C03632=1090.259,178.898,430.027,176.034,19.768,152.995
C03633=1090.254,178.648,430.050,176.031,19.767,152.995
C03634=1090.248,178.399,430.073,176.028,19.766,152.995
C03635=1090.242,178.150,430.094,176.025,19.765,152.995
C03636=1090.237,177.901,430.116,176.023,19.764,152.995
C03637=1090.232,177.652,430.139,176.020,19.763,152.996
C03638=1090.225,177.403,430.161,176.017,19.762,152.996
C03639=1090.220,177.155,430.183,176.014,19.761,152.996
C03640=1090.215,176.906,430.206,176.012,19.760,152.997
C03641=1090.209,176.656,430.227,176.009,19.759,152.997
C03642=1090.203,176.407,430.250,176.006,19.758,152.997
C03643=1090.197,176.131,430.274,176.003,19.756,152.997
C03644=1090.191,175.854,430.299,176.001,19.755,152.997
C03645=1090.184,175.577,430.323,175.997,19.753,152.998
C03646=1090.178,175.300,430.348,175.994,19.752,152.998
C03647=1090.172,175.051,430.370,175.992,19.751,152.998
C03648=1090.167,174.803,430.393,175.989,19.750,152.998
C03649=1090.162,174.553,430.415,175.986,19.749,152.999
C03650=1090.155,174.304,430.437,175.983,19.748,152.999
C03651=1090.151,174.055,430.458,175.981,19.747,152.999
C03652=1090.144,173.806,430.481,175.978,19.746,152.999
C03653=1090.139,173.557,430.503,175.975,19.745,153.000
C03654=1090.134,173.308,430.525,175.972,19.744,153.000
C03655=1090.128,173.059,430.546,175.970,19.742,153.000
C03656=1090.123,172.811,430.569,175.967,19.741,153.000
C03657=1090.116,172.561,430.591,175.965,19.740,153.000
C03658=1090.111,172.312,430.613,175.962,19.739,153.001
C03659=1090.106,172.063,430.634,175.960,19.738,153.001
C03660=1090.100,171.814,430.656,175.957,19.737,153.001
C03661=1090.095,171.565,430.678,175.954,19.736,153.001
C03662=1090.089,171.317,430.701,175.952,19.734,153.001
C03663=1090.084,171.068,430.722,175.949,19.733,153.002
C03664=1090.078,170.819,430.744,175.946,19.732,153.002
C03665=1090.073,170.570,430.766,175.943,19.731,153.002
C03666=1090.067,170.321,430.788,175.941,19.730,153.002
C03667=1090.061,170.071,430.810,175.938,19.729,153.003
C03668=1090.056,169.822,430.831,175.935,19.728,153.003
C03669=1090.050,169.573,430.853,175.933,19.726,153.003
C03670=1090.045,169.324,430.875,175.930,19.725,153.003
C03671=1090.039,169.076,430.898,175.927,19.724,153.004
C03672=1090.034,168.827,430.919,175.925,19.722,153.004
C03673=1090.028,168.578,430.941,175.923,19.722,153.004
C03674=1090.023,168.329,430.962,175.920,19.720,153.004
C03675=1090.017,168.080,430.985,175.917,19.719,153.004
C03676=1090.012,167.831,431.006,175.915,19.718,153.004
C03677=1090.006,167.582,431.028,175.912,19.717,153.005
C03678=1090.001,167.333,431.049,175.909,19.716,153.005
C03679=1089.995,167.083,431.072,175.906,19.715,153.005
C03680=1089.990,166.835,431.093,175.904,19.713,153.005
C03681=1089.984,166.586,431.114,175.901,19.712,153.005
C03682=1089.979,166.336,431.136,175.899,19.711,153.006
C03683=1089.973,166.088,431.157,175.896,19.710,153.006
C03684=1089.968,165.838,431.179,175.893,19.708,153.006
C03685=1089.962,165.590,431.200,175.891,19.707,153.006
C03686=1089.957,165.340,431.223,175.889,19.707,153.006
C03687=1089.951,165.092,431.244,175.886,19.705,153.007
C03688=1089.946,164.842,431.266,175.883,19.704,153.007
C03689=1089.940,164.594,431.287,175.881,19.702,153.007
C03690=1089.935,164.345,431.309,175.878,19.701,153.007
C03691=1089.930,164.095,431.330,175.875,19.700,153.007
C03692=1089.924,163.847,431.351,175.873,19.699,153.008
C03693=1089.919,163.597,431.374,175.870,19.697,153.008
C03694=1089.913,163.349,431.395,175.867,19.696,153.008
C03695=1089.908,163.100,431.416,175.865,19.695,153.008
C03696=1089.902,162.851,431.438,175.863,19.694,153.008
C03697=1089.897,162.601,431.459,175.860,19.693,153.008
C03698=1089.892,162.353,431.481,175.858,19.692,153.009
C03699=1089.886,162.103,431.502,175.855,19.690,153.009
C03700=1089.880,161.855,431.524,175.852,19.689,153.009
C03701=1089.876,161.606,431.545,175.850,19.688,153.009
C03702=1089.870,161.356,431.567,175.847,19.687,153.009
C03703=1089.864,161.108,431.588,175.844,19.685,153.010
C03704=1089.858,160.858,431.609,175.842,19.684,153.010
C03705=1089.853,160.609,431.630,175.840,19.683,153.010
C03706=1089.847,160.360,431.652,175.837,19.682,153.010
C03707=1089.841,160.083,431.676,175.834,19.680,153.010
C03708=1089.835,159.806,431.700,175.831,19.679,153.011
C03709=1089.829,159.528,431.723,175.828,19.678,153.011
C03710=1089.822,159.251,431.747,175.825,19.677,153.011
C03711=1089.817,159.002,431.768,175.823,19.675,153.011
C03712=1089.811,158.754,431.789,175.820,19.674,153.011
C03713=1089.806,158.504,431.810,175.818,19.673,153.012
C03714=1089.800,158.255,431.831,175.815,19.672,153.012
C03715=1089.794,158.005,431.852,175.813,19.671,153.012
C03716=1089.789,157.757,431.873,175.810,19.670,153.012
C03717=1089.783,157.508,431.895,175.808,19.668,153.012
C03718=1089.777,157.259,431.916,175.805,19.667,153.013
C03719=1089.772,157.010,431.937,175.802,19.666,153.013
C03720=1089.767,156.761,431.958,175.800,19.664,153.013
C03721=1089.761,156.511,431.980,175.797,19.663,153.013
C03722=1089.756,156.262,432.000,175.795,19.662,153.013
C03723=1089.750,156.014,432.021,175.793,19.661,153.013
C03724=1089.744,155.764,432.042,175.790,19.660,153.014
C03725=1089.739,155.516,432.064,175.787,19.658,153.014
C03726=1089.733,155.266,432.084,175.785,19.657,153.014
C03727=1089.727,155.017,432.106,175.782,19.656,153.014
C03728=1089.722,154.768,432.126,175.779,19.655,153.014
C03729=1089.716,154.520,432.148,175.778,19.654,153.015
C03730=1089.711,154.270,432.169,175.775,19.653,153.015
C03731=1089.705,154.021,432.190,175.772,19.651,153.015
C03732=1089.700,153.772,432.210,175.769,19.650,153.015
C03733=1089.694,153.524,432.232,175.767,19.649,153.015
C03734=1089.688,153.274,432.253,175.764,19.648,153.016
C03735=1089.682,153.025,432.273,175.762,19.647,153.016
C03736=1089.677,152.776,432.294,175.760,19.646,153.016
C03737=1089.671,152.527,432.315,175.757,19.644,153.016
C03738=1089.666,152.278,432.335,175.755,19.642,153.016
C03739=1089.660,152.029,432.357,175.752,19.641,153.016
C03740=1089.655,151.780,432.377,175.749,19.640,153.017
C03741=1089.649,151.530,432.398,175.747,19.639,153.017
C03742=1089.643,151.282,432.419,175.745,19.638,153.017
C03743=1089.638,151.032,432.440,175.742,19.636,153.017
C03744=1089.633,150.783,432.460,175.739,19.635,153.017
C03745=1089.627,150.534,432.482,175.737,19.634,153.017
C03746=1089.621,150.285,432.502,175.734,19.633,153.018
C03747=1089.615,150.036,432.523,175.732,19.632,153.018
C03748=1089.610,149.788,432.544,175.730,19.630,153.018
C03749=1089.605,149.539,432.564,175.727,19.629,153.018
C03750=1089.599,149.289,432.585,175.725,19.628,153.018
C03751=1089.594,149.040,432.606,175.722,19.626,153.018
C03752=1089.588,148.791,432.627,175.719,19.625,153.019
C03753=1089.582,148.542,432.647,175.718,19.624,153.019
C03754=1089.576,148.292,432.668,175.715,19.623,153.019
C03755=1089.571,148.043,432.689,175.712,19.622,153.019
C03756=1089.566,147.794,432.709,175.710,19.620,153.019
C03757=1089.559,147.546,432.730,175.707,19.619,153.020
C03758=1089.554,147.297,432.750,175.705,19.618,153.020
C03759=1089.548,147.047,432.771,175.703,19.616,153.020
C03760=1089.543,146.798,432.792,175.700,19.615,153.020
C03761=1089.537,146.549,432.812,175.697,19.614,153.020
C03762=1089.532,146.300,432.832,175.695,19.613,153.020
C03763=1089.526,146.051,432.853,175.693,19.612,153.020
C03764=1089.520,145.801,432.873,175.690,19.610,153.021
C03765=1089.514,145.553,432.895,175.688,19.609,153.021
C03766=1089.509,145.304,432.915,175.685,19.608,153.021
C03767=1089.504,145.055,432.936,175.683,19.606,153.021
C03768=1089.498,144.806,432.956,175.681,19.606,153.021
C03769=1089.493,144.557,432.976,175.678,19.604,153.021
C03770=1089.487,144.307,432.997,175.676,19.603,153.022
C03771=1089.480,144.030,433.019,175.673,19.601,153.022
C03772=1089.474,143.752,433.042,175.670,19.600,153.022
C03773=1089.468,143.475,433.065,175.668,19.599,153.022
C03774=1089.462,143.197,433.088,175.665,19.597,153.022
C03775=1089.456,142.948,433.108,175.662,19.596,153.022
C03776=1089.451,142.699,433.128,175.660,19.594,153.023
C03777=1089.445,142.450,433.149,175.657,19.593,153.023
C03778=1089.439,142.201,433.169,175.655,19.591,153.023
C03779=1089.434,141.951,433.190,175.653,19.591,153.023
C03780=1089.428,141.702,433.210,175.650,19.589,153.023
C03781=1089.422,141.453,433.230,175.648,19.588,153.023
C03782=1089.417,141.204,433.251,175.645,19.586,153.023
C03783=1089.412,140.955,433.271,175.643,19.585,153.024
C03784=1089.406,140.706,433.291,175.641,19.584,153.024
C03785=1089.401,140.457,433.311,175.638,19.583,153.024
C03786=1089.395,140.208,433.331,175.636,19.581,153.024
C03787=1089.390,139.959,433.352,175.633,19.580,153.024
C03788=1089.384,139.710,433.371,175.631,19.579,153.024
C03789=1089.378,139.461,433.392,175.629,19.578,153.024
C03790=1089.372,139.211,433.412,175.626,19.576,153.025
C03791=1089.366,138.962,433.433,175.624,19.575,153.025
C03792=1089.361,138.713,433.452,175.622,19.574,153.025
C03793=1089.356,138.463,433.473,175.619,19.573,153.025
C03794=1089.350,138.215,433.493,175.617,19.571,153.025
C03795=1089.344,137.966,433.513,175.614,19.570,153.025
C03796=1089.338,137.717,433.533,175.611,19.568,153.025
C03797=1089.333,137.467,433.553,175.610,19.567,153.026
C03798=1089.327,137.218,433.573,175.607,19.566,153.026
C03799=1089.322,136.969,433.594,175.604,19.564,153.026
C03800=1089.316,136.720,433.613,175.602,19.563,153.026
C03801=1089.310,136.471,433.633,175.600,19.562,153.026
C03802=1089.305,136.222,433.653,175.598,19.560,153.026
C03803=1089.299,135.973,433.673,175.595,19.559,153.026
C03804=1089.294,135.724,433.694,175.592,19.558,153.027
C03805=1089.288,135.474,433.713,175.591,19.557,153.027
C03806=1089.283,135.225,433.734,175.588,19.555,153.027
C03807=1089.277,134.976,433.754,175.586,19.554,153.027
C03808=1089.271,134.727,433.773,175.583,19.552,153.027
C03809=1089.266,134.478,433.793,175.581,19.551,153.027
C03810=1089.260,134.229,433.813,175.579,19.550,153.027
C03811=1089.254,133.980,433.833,175.576,19.548,153.027
C03812=1089.249,133.730,433.853,175.574,19.547,153.028
C03813=1089.243,133.482,433.873,175.572,19.546,153.028
C03814=1089.238,133.232,433.893,175.569,19.545,153.028
C03815=1089.232,132.983,433.913,175.567,19.543,153.028
C03816=1089.226,132.734,433.932,175.565,19.542,153.028
C03817=1089.221,132.485,433.953,175.562,19.541,153.028
C03818=1089.215,132.236,433.973,175.560,19.539,153.028
C03819=1089.210,131.986,433.992,175.557,19.537,153.029
C03820=1089.204,131.737,434.012,175.556,19.536,153.029
C03821=1089.199,131.488,434.032,175.553,19.535,153.029
C03822=1089.193,131.239,434.052,175.550,19.534,153.029
C03823=1089.187,130.989,434.071,175.548,19.532,153.029
C03824=1089.181,130.741,434.091,175.546,19.531,153.029
C03825=1089.175,130.491,434.110,175.544,19.530,153.029
C03826=1089.170,130.242,434.131,175.541,19.528,153.029
C03827=1089.164,129.993,434.150,175.539,19.527,153.030
C03828=1089.158,129.744,434.170,175.537,19.526,153.030
C03829=1089.153,129.494,434.189,175.534,19.524,153.030
C03830=1089.147,129.246,434.209,175.532,19.523,153.030
C03831=1089.141,128.996,434.228,175.530,19.522,153.030
C03832=1089.135,128.747,434.248,175.527,19.521,153.030
C03833=1089.130,128.498,434.268,175.525,19.519,153.030
C03834=1089.125,128.250,434.288,175.522,19.518,153.031
C03835=1089.118,127.971,434.309,175.520,19.516,153.031
C03836=1089.112,127.694,434.331,175.517,19.515,153.031
C03837=1089.105,127.416,434.353,175.515,19.513,153.031
C03838=1089.099,127.138,434.375,175.512,19.512,153.031
C03839=1089.094,126.889,434.394,175.510,19.511,153.031
C03840=1089.088,126.640,434.414,175.508,19.509,153.031
C03841=1089.082,126.391,434.433,175.505,19.507,153.031
C03842=1089.076,126.141,434.453,175.504,19.506,153.031
C03843=1089.070,125.892,434.473,175.501,19.505,153.032
C03844=1089.065,125.644,434.491,175.499,19.503,153.032
C03845=1089.059,125.394,434.511,175.496,19.502,153.032
C03846=1089.053,125.146,434.531,175.494,19.501,153.032
C03847=1089.048,124.896,434.550,175.492,19.499,153.032
C03848=1089.043,124.646,434.570,175.489,19.498,153.032
C03849=1089.037,124.397,434.589,175.488,19.497,153.032
C03850=1089.031,124.148,434.609,175.485,19.495,153.032
C03851=1089.026,123.899,434.628,175.482,19.494,153.033
C03852=1089.020,123.650,434.647,175.481,19.493,153.033
C03853=1089.015,123.400,434.666,175.478,19.491,153.033
C03854=1089.009,123.152,434.686,175.476,19.489,153.033
C03855=1089.003,122.902,434.705,175.473,19.488,153.033
C03856=1088.997,122.653,434.725,175.472,19.487,153.033
C03857=1088.992,122.404,434.744,175.469,19.485,153.033
C03858=1088.986,122.155,434.764,175.467,19.484,153.033
C03859=1088.981,121.906,434.783,175.465,19.483,153.033
C03860=1088.975,121.656,434.802,175.462,19.481,153.033
C03861=1088.969,121.407,434.821,175.460,19.480,153.034
C03862=1088.964,121.158,434.840,175.458,19.479,153.034
C03863=1088.958,120.909,434.859,175.456,19.477,153.034
C03864=1088.953,120.659,434.879,175.453,19.475,153.034
C03865=1088.947,120.411,434.899,175.452,19.474,153.034
C03866=1088.942,120.162,434.917,175.449,19.472,153.034
C03867=1088.936,119.912,434.937,175.447,19.471,153.034
C03868=1088.930,119.663,434.956,175.445,19.470,153.034
C03869=1088.925,119.414,434.975,175.443,19.468,153.034
C03870=1088.919,119.165,434.994,175.440,19.466,153.034
C03871=1088.914,118.915,435.013,175.438,19.465,153.034
C03872=1088.908,118.666,435.033,175.436,19.464,153.034
C03873=1088.902,118.416,435.052,175.433,19.462,153.035
C03874=1088.897,118.168,435.071,175.431,19.460,153.035
C03875=1088.892,117.918,435.090,175.429,19.459,153.035
C03876=1088.886,117.669,435.109,175.427,19.458,153.035
C03877=1088.881,117.420,435.128,175.424,19.456,153.035
C03878=1088.875,117.171,435.147,175.423,19.455,153.035
C03879=1088.869,116.921,435.167,175.420,19.453,153.035
C03880=1088.864,116.673,435.185,175.418,19.452,153.035
C03881=1088.859,116.423,435.205,175.416,19.451,153.035
C03882=1088.853,116.174,435.224,175.414,19.449,153.035
C03883=1088.848,115.925,435.243,175.411,19.447,153.035
C03884=1088.842,115.676,435.262,175.409,19.446,153.035
C03885=1088.837,115.426,435.281,175.407,19.445,153.036
C03886=1088.831,115.177,435.300,175.405,19.443,153.036
C03887=1088.825,114.928,435.319,175.403,19.442,153.036
C03888=1088.819,114.679,435.338,175.400,19.440,153.036
C03889=1088.814,114.430,435.357,175.398,19.438,153.036
C03890=1088.809,114.181,435.376,175.396,19.437,153.036
C03891=1088.803,113.931,435.395,175.394,19.435,153.036
C03892=1088.798,113.682,435.414,175.391,19.434,153.036
C03893=1088.792,113.433,435.432,175.390,19.432,153.036
C03894=1088.786,113.183,435.451,175.387,19.431,153.036
C03895=1088.780,112.934,435.471,175.386,19.430,153.036
C03896=1088.775,112.685,435.490,175.383,19.428,153.036
C03897=1088.769,112.436,435.508,175.381,19.426,153.036
C03898=1088.763,112.186,435.527,175.379,19.425,153.036
C03899=1088.757,111.908,435.548,175.377,19.424,153.037
C03900=1088.751,111.631,435.569,175.374,19.422,153.037
C03901=1088.745,111.353,435.590,175.372,19.420,153.037
C03902=1088.738,111.076,435.611,175.369,19.419,153.037
C03903=1088.733,110.827,435.630,175.367,19.417,153.037
C03904=1088.727,110.578,435.648,175.365,19.416,153.037
C03905=1088.722,110.328,435.667,175.363,19.414,153.037
C03906=1088.716,110.079,435.685,175.360,19.413,153.037
C03907=1088.710,109.830,435.704,175.358,19.412,153.037
C03908=1088.704,109.580,435.723,175.356,19.410,153.037
C03909=1088.699,109.331,435.741,175.354,19.408,153.037
C03910=1088.693,109.082,435.760,175.352,19.407,153.037
C03911=1088.687,108.833,435.780,175.350,19.405,153.037
C03912=1088.682,108.584,435.797,175.347,19.403,153.038
C03913=1088.676,108.334,435.816,175.345,19.402,153.038
C03914=1088.670,108.085,435.835,175.343,19.400,153.038
C03915=1088.665,107.836,435.853,175.341,19.399,153.038
C03916=1088.659,107.586,435.872,175.339,19.398,153.038
C03917=1088.653,107.338,435.891,175.337,19.396,153.038
C03918=1088.648,107.088,435.909,175.335,19.395,153.038
C03919=1088.642,106.839,435.928,175.332,19.393,153.038
C03920=1088.637,106.590,435.947,175.330,19.391,153.038
C03921=1088.630,106.340,435.965,175.328,19.390,153.038
C03922=1088.625,106.091,435.984,175.326,19.388,153.038
C03923=1088.619,105.842,436.001,175.324,19.387,153.038
C03924=1088.614,105.593,436.020,175.322,19.386,153.038
C03925=1088.609,105.343,436.039,175.320,19.384,153.038
C03926=1088.603,105.094,436.057,175.318,19.383,153.038
C03927=1088.597,104.845,436.076,175.316,19.381,153.038
C03928=1088.591,104.595,436.094,175.313,19.379,153.039
C03929=1088.586,104.347,436.113,175.311,19.378,153.039
C03930=1088.580,104.097,436.131,175.309,19.376,153.039
C03931=1088.575,103.848,436.150,175.307,19.375,153.039
C03932=1088.569,103.598,436.168,175.305,19.373,153.039
C03933=1088.564,103.350,436.187,175.303,19.371,153.039
C03934=1088.558,103.100,436.205,175.301,19.370,153.039
C03935=1088.552,102.851,436.224,175.299,19.368,153.039
C03936=1088.546,102.601,436.242,175.297,19.367,153.039
C03937=1088.541,102.353,436.260,175.295,19.365,153.039
C03938=1088.535,102.103,436.278,175.292,19.364,153.039
C03939=1088.530,101.854,436.297,175.291,19.362,153.039
C03940=1088.524,101.604,436.315,175.288,19.361,153.039
C03941=1088.519,101.355,436.333,175.287,19.359,153.039
C03942=1088.513,101.106,436.352,175.284,19.358,153.039
C03943=1088.508,100.857,436.370,175.282,19.356,153.039
C03944=1088.502,100.607,436.388,175.280,19.355,153.039
C03945=1088.496,100.358,436.406,175.278,19.353,153.039
C03946=1088.491,100.108,436.425,175.276,19.352,153.039
C03947=1088.485,99.860,436.443,175.274,19.350,153.039
C03948=1088.479,99.610,436.461,175.271,19.348,153.040
C03949=1088.474,99.361,436.479,175.270,19.347,153.040
C03950=1088.467,99.112,436.498,175.267,19.345,153.040
C03951=1088.462,98.863,436.515,175.266,19.344,153.040
C03952=1088.457,98.613,436.534,175.263,19.342,153.040
C03953=1088.451,98.364,436.552,175.261,19.341,153.040
C03954=1088.445,98.114,436.570,175.259,19.339,153.040
C03955=1088.439,97.865,436.588,175.257,19.337,153.040
C03956=1088.433,97.616,436.607,175.255,19.336,153.040
C03957=1088.428,97.367,436.625,175.253,19.334,153.040
C03958=1088.422,97.117,436.643,175.250,19.332,153.040
C03959=1088.417,96.868,436.661,175.249,19.331,153.040
C03960=1088.411,96.619,436.679,175.247,19.329,153.040
C03961=1088.405,96.370,436.697,175.245,19.328,153.040
C03962=1088.400,96.121,436.714,175.243,19.326,153.040
C03963=1088.393,95.843,436.735,175.240,19.324,153.040
C03964=1088.387,95.565,436.755,175.238,19.323,153.040
C03965=1088.381,95.288,436.775,175.235,19.321,153.040
C03966=1088.375,95.010,436.795,175.234,19.319,153.040
C03967=1088.369,94.760,436.814,175.231,19.318,153.040
C03968=1088.363,94.511,436.831,175.229,19.316,153.040
C03969=1088.358,94.262,436.849,175.227,19.315,153.040
C03970=1088.352,94.013,436.867,175.225,19.313,153.040
C03971=1088.346,93.764,436.885,175.223,19.312,153.041
C03972=1088.341,93.514,436.903,175.221,19.310,153.041
C03973=1088.335,93.265,436.921,175.220,19.308,153.040
C03974=1088.329,93.016,436.939,175.217,19.307,153.041
C03975=1088.323,92.766,436.957,175.215,19.305,153.041
C03976=1088.319,92.517,436.975,175.213,19.303,153.041
C03977=1088.313,92.268,436.993,175.211,19.301,153.041
C03978=1088.307,92.018,437.011,175.209,19.300,153.041
C03979=1088.301,91.769,437.028,175.207,19.298,153.041
C03980=1088.296,91.520,437.046,175.205,19.297,153.041
C03981=1088.291,91.270,437.064,175.203,19.295,153.041
C03982=1088.285,91.021,437.082,175.201,19.293,153.041
C03983=1088.280,90.772,437.099,175.199,19.292,153.041
C03984=1088.273,90.522,437.117,175.197,19.290,153.041
C03985=1088.268,90.273,437.135,175.195,19.289,153.041
C03986=1088.262,90.024,437.152,175.193,19.287,153.041
C03987=1088.256,89.774,437.170,175.191,19.286,153.041
C03988=1088.251,89.525,437.188,175.189,19.284,153.041
C03989=1088.245,89.276,437.206,175.187,19.282,153.041
C03990=1088.239,89.027,437.223,175.185,19.281,153.041
C03991=1088.234,88.778,437.241,175.183,19.279,153.041
C03992=1088.227,88.528,437.259,175.181,19.278,153.041
C03993=1088.222,88.279,437.276,175.179,19.276,153.041
C03994=1088.216,88.030,437.294,175.177,19.274,153.041
C03995=1088.210,87.780,437.312,175.175,19.273,153.041
C03996=1088.205,87.531,437.330,175.173,19.271,153.041
C03997=1088.199,87.282,437.347,175.171,19.269,153.041
C03998=1088.193,87.032,437.365,175.169,19.268,153.041
C03999=1088.188,86.783,437.383,175.167,19.266,153.041
C04000=1088.182,86.534,437.400,175.165,19.264,153.041
C04001=1088.176,86.284,437.418,175.163,19.263,153.041
C04002=1088.170,86.035,437.436,175.161,19.261,153.041
C04003=1088.165,85.786,437.452,175.159,19.259,153.041
C04004=1088.160,85.537,437.470,175.157,19.258,153.041
C04005=1088.154,85.287,437.488,175.155,19.256,153.041
C04006=1088.148,85.038,437.506,175.153,19.254,153.041
C04007=1088.143,84.789,437.523,175.152,19.253,153.041
C04008=1088.136,84.539,437.541,175.149,19.251,153.041
C04009=1088.131,84.289,437.558,175.148,19.250,153.041
C04010=1088.126,84.040,437.575,175.145,19.248,153.041
C04011=1088.120,83.791,437.593,175.143,19.246,153.041
C04012=1088.114,83.542,437.611,175.141,19.245,153.041
C04013=1088.109,83.292,437.629,175.139,19.243,153.041
C04014=1088.103,83.043,437.645,175.138,19.241,153.041
C04015=1088.097,82.794,437.662,175.135,19.239,153.041
C04016=1088.091,82.544,437.680,175.134,19.238,153.041
C04017=1088.085,82.295,437.698,175.131,19.236,153.041
C04018=1088.080,82.046,437.715,175.130,19.234,153.041
C04019=1088.075,81.797,437.732,175.128,19.232,153.041
C04020=1088.069,81.548,437.750,175.126,19.231,153.041
C04021=1088.063,81.298,437.768,175.124,19.229,153.041
C04022=1088.058,81.048,437.785,175.122,19.228,153.041
C04023=1088.052,80.799,437.802,175.120,19.226,153.041
C04024=1088.047,80.550,437.820,175.118,19.224,153.041
C04025=1088.041,80.301,437.836,175.116,19.222,153.041
C04026=1088.035,80.051,437.854,175.114,19.221,153.041
C04027=1088.029,79.774,437.874,175.112,19.219,153.041
C04028=1088.023,79.496,437.892,175.110,19.217,153.041
C04029=1088.016,79.218,437.912,175.108,19.215,153.041
C04030=1088.010,78.941,437.931,175.105,19.213,153.041
C04031=1088.005,78.692,437.948,175.104,19.212,153.041
C04032=1087.999,78.442,437.965,175.102,19.210,153.041
C04033=1087.994,78.193,437.983,175.100,19.209,153.041
C04034=1087.987,77.944,438.000,175.098,19.206,153.041
C04035=1087.982,77.694,438.017,175.096,19.205,153.041
C04036=1087.976,77.445,438.035,175.094,19.203,153.041
C04037=1087.970,77.196,438.051,175.092,19.201,153.041
C04038=1087.965,76.947,438.068,175.090,19.199,153.041
C04039=1087.959,76.696,438.086,175.088,19.198,153.041
C04040=1087.953,76.447,438.103,175.086,19.196,153.041
C04041=1087.948,76.198,438.119,175.085,19.195,153.041
C04042=1087.942,75.949,438.137,175.082,19.193,153.041
C04043=1087.936,75.700,438.155,175.081,19.191,153.041
C04044=1087.931,75.451,438.171,175.078,19.190,153.041
C04045=1087.924,75.201,438.189,175.077,19.188,153.041
C04046=1087.919,74.951,438.206,175.075,19.186,153.041
C04047=1087.913,74.702,438.223,175.073,19.185,153.041
C04048=1087.908,74.453,438.239,175.071,19.183,153.041
C04049=1087.903,74.203,438.256,175.069,19.181,153.041
C04050=1087.896,73.954,438.273,175.067,19.179,153.041
C04051=1087.891,73.705,438.290,175.066,19.178,153.041
C04052=1087.886,73.456,438.308,175.063,19.176,153.041
C04053=1087.879,73.206,438.324,175.062,19.174,153.041
C04054=1087.873,72.957,438.342,175.060,19.172,153.041
C04055=1087.868,72.707,438.359,175.058,19.171,153.041
C04056=1087.862,72.458,438.375,175.056,19.169,153.041
C04057=1087.857,72.209,438.392,175.054,19.167,153.041
C04058=1087.851,71.959,438.409,175.052,19.165,153.041
C04059=1087.845,71.710,438.426,175.051,19.164,153.041
C04060=1087.840,71.460,438.443,175.048,19.162,153.041
C04061=1087.834,71.211,438.459,175.047,19.160,153.041
C04062=1087.829,70.962,438.477,175.044,19.159,153.041
C04063=1087.823,70.713,438.493,175.043,19.157,153.041
C04064=1087.817,70.463,438.510,175.041,19.155,153.041
C04065=1087.812,70.214,438.528,175.039,19.154,153.041
C04066=1087.805,69.964,438.544,175.037,19.152,153.041
C04067=1087.800,69.714,438.561,175.035,19.150,153.041
C04068=1087.794,69.466,438.578,175.033,19.148,153.041
C04069=1087.789,69.216,438.595,175.032,19.147,153.041
C04070=1087.783,68.967,438.611,175.029,19.144,153.041
C04071=1087.777,68.718,438.629,175.028,19.143,153.041
C04072=1087.771,68.468,438.645,175.026,19.141,153.041
C04073=1087.766,68.219,438.662,175.024,19.139,153.041
C04074=1087.760,67.969,438.678,175.022,19.137,153.041
C04075=1087.755,67.720,438.696,175.021,19.136,153.041
C04076=1087.749,67.471,438.712,175.018,19.134,153.041
C04077=1087.743,67.221,438.729,175.017,19.133,153.041
C04078=1087.738,66.972,438.745,175.014,19.131,153.041
C04079=1087.732,66.722,438.762,175.013,19.129,153.041
C04080=1087.726,66.473,438.779,175.011,19.127,153.041
C04081=1087.720,66.224,438.795,175.009,19.126,153.041
C04082=1087.715,65.974,438.812,175.007,19.124,153.041
C04083=1087.709,65.725,438.828,175.005,19.122,153.041
C04084=1087.704,65.475,438.845,175.003,19.120,153.041
C04085=1087.697,65.227,438.862,175.002,19.119,153.041
C04086=1087.692,64.977,438.879,174.999,19.116,153.041
C04087=1087.686,64.728,438.895,174.998,19.115,153.041
C04088=1087.680,64.478,438.911,174.996,19.113,153.041
C04089=1087.675,64.229,438.928,174.994,19.111,153.041
C04090=1087.669,63.979,438.945,174.993,19.110,153.040
C04091=1087.662,63.701,438.963,174.990,19.108,153.040
C04092=1087.655,63.424,438.981,174.988,19.106,153.040
C04093=1087.649,63.146,439.000,174.986,19.104,153.040
C04094=1087.643,62.869,439.018,174.984,19.102,153.040
C04095=1087.637,62.620,439.034,174.982,19.100,153.040
C04096=1087.631,62.370,439.051,174.981,19.099,153.040
C04097=1087.626,62.121,439.068,174.978,19.097,153.040
C04098=1087.620,61.871,439.084,174.977,19.095,153.040
C04099=1087.614,61.622,439.100,174.975,19.093,153.040
C04100=1087.608,61.373,439.116,174.973,19.092,153.040
C04101=1087.603,61.123,439.133,174.971,19.090,153.040
C04102=1087.597,60.874,439.149,174.970,19.088,153.040
C04103=1087.591,60.624,439.166,174.968,19.086,153.040
C04104=1087.585,60.375,439.182,174.966,19.084,153.040
C04105=1087.579,60.125,439.198,174.964,19.083,153.040
C04106=1087.574,59.876,439.215,174.962,19.081,153.040
C04107=1087.568,59.626,439.231,174.961,19.079,153.040
C04108=1087.562,59.377,439.248,174.958,19.077,153.040
C04109=1087.556,59.128,439.264,174.957,19.076,153.040
C04110=1087.550,58.878,439.280,174.955,19.074,153.040
C04111=1087.545,58.629,439.297,174.953,19.072,153.040
C04112=1087.539,58.379,439.313,174.951,19.070,153.040
C04113=1087.533,58.130,439.329,174.949,19.069,153.040
C04114=1087.527,57.881,439.346,174.948,19.067,153.040
C04115=1087.521,57.631,439.362,174.946,19.065,153.040
C04116=1087.515,57.382,439.378,174.944,19.064,153.040
C04117=1087.510,57.132,439.395,174.942,19.061,153.040
C04118=1087.504,56.883,439.411,174.941,19.060,153.040
C04119=1087.499,56.634,439.426,174.938,19.058,153.040
C04120=1087.493,56.384,439.443,174.937,19.056,153.040
C04121=1087.487,56.135,439.459,174.935,19.054,153.040
C04122=1087.481,55.886,439.475,174.933,19.053,153.040
C04123=1087.475,55.636,439.492,174.932,19.051,153.040
C04124=1087.469,55.387,439.508,174.929,19.049,153.040
C04125=1087.464,55.137,439.525,174.928,19.048,153.040
C04126=1087.458,54.887,439.540,174.926,19.046,153.040
C04127=1087.452,54.638,439.556,174.925,19.044,153.039
C04128=1087.447,54.389,439.572,174.922,19.042,153.039
C04129=1087.441,54.140,439.589,174.921,19.040,153.039
C04130=1087.435,53.891,439.605,174.919,19.038,153.039
C04131=1087.429,53.641,439.620,174.917,19.037,153.039
C04132=1087.423,53.391,439.637,174.916,19.035,153.039
C04133=1087.418,53.142,439.653,174.913,19.033,153.039
C04134=1087.413,52.893,439.669,174.912,19.031,153.039
C04135=1087.407,52.643,439.685,174.910,19.029,153.039
C04136=1087.401,52.394,439.701,174.908,19.027,153.039
C04137=1087.395,52.144,439.717,174.906,19.025,153.039
C04138=1087.389,51.895,439.734,174.905,19.024,153.039
C04139=1087.384,51.645,439.749,174.903,19.022,153.039
C04140=1087.378,51.396,439.765,174.901,19.020,153.039
C04141=1087.372,51.147,439.781,174.900,19.019,153.039
C04142=1087.367,50.897,439.797,174.898,19.016,153.039
C04143=1087.361,50.648,439.813,174.896,19.015,153.039
C04144=1087.355,50.398,439.829,174.894,19.013,153.039
C04145=1087.350,50.149,439.845,174.892,19.011,153.039
C04146=1087.345,49.899,439.861,174.891,19.010,153.038
C04147=1087.339,49.650,439.878,174.889,19.007,153.038
C04148=1087.333,49.400,439.893,174.887,19.005,153.038
C04149=1087.328,49.152,439.909,174.885,19.003,153.038
C04150=1087.322,48.902,439.925,174.884,19.002,153.038
C04151=1087.316,48.652,439.941,174.881,19.000,153.038
C04152=1087.310,48.403,439.957,174.880,18.998,153.038
C04153=1087.305,48.154,439.972,174.879,18.996,153.038
C04154=1087.299,47.904,439.989,174.877,18.994,153.038
C04155=1087.292,47.626,440.006,174.875,18.993,153.038
C04156=1087.287,47.348,440.024,174.873,18.991,153.038
C04157=1087.281,47.070,440.041,174.871,18.988,153.038
C04158=1087.274,46.793,440.059,174.869,18.986,153.038
C04159=1087.268,46.543,440.075,174.867,18.985,153.038
C04160=1087.262,46.294,440.091,174.866,18.982,153.038
C04161=1087.257,46.044,440.106,174.864,18.980,153.038
C04162=1087.251,45.795,440.122,174.862,18.979,153.037
C04163=1087.245,45.545,440.138,174.860,18.977,153.037
C04164=1087.240,45.296,440.154,174.859,18.975,153.037
C04165=1087.234,45.047,440.169,174.857,18.973,153.037
C04166=1087.228,44.797,440.186,174.855,18.971,153.037
C04167=1087.223,44.548,440.201,174.854,18.969,153.037
C04168=1087.217,44.299,440.217,174.852,18.967,153.037
C04169=1087.212,44.049,440.233,174.850,18.966,153.037
C04170=1087.206,43.800,440.248,174.849,18.964,153.037
C04171=1087.201,43.550,440.264,174.847,18.962,153.037
C04172=1087.195,43.300,440.280,174.845,18.960,153.037
C04173=1087.189,43.051,440.296,174.843,18.958,153.037
C04174=1087.183,42.802,440.310,174.841,18.956,153.037
C04175=1087.177,42.552,440.327,174.840,18.955,153.037
C04176=1087.172,42.302,440.342,174.838,18.952,153.037
C04177=1087.167,42.054,440.358,174.837,18.951,153.036
C04178=1087.161,41.804,440.374,174.834,18.949,153.036
C04179=1087.154,41.554,440.389,174.833,18.947,153.036
C04180=1087.149,41.305,440.404,174.831,18.946,153.036
C04181=1087.143,41.055,440.420,174.829,18.943,153.036
C04182=1087.138,40.806,440.436,174.828,18.942,153.036
C04183=1087.132,40.557,440.451,174.826,18.940,153.036
C04184=1087.126,40.307,440.466,174.824,18.938,153.036
C04185=1087.120,40.057,440.482,174.823,18.936,153.036
C04186=1087.115,39.809,440.498,174.821,18.934,153.036
C04187=1087.109,39.559,440.513,174.819,18.932,153.036
C04188=1087.103,39.309,440.528,174.817,18.930,153.036
C04189=1087.098,39.060,440.544,174.816,18.928,153.036
C04190=1087.092,38.810,440.560,174.814,18.927,153.036
C04191=1087.086,38.560,440.575,174.812,18.925,153.036
C04192=1087.080,38.312,440.591,174.811,18.923,153.036
C04193=1087.075,38.062,440.606,174.809,18.921,153.035
C04194=1087.070,37.813,440.621,174.807,18.919,153.035
C04195=1087.064,37.563,440.637,174.806,18.918,153.035
C04196=1087.057,37.314,440.652,174.804,18.916,153.035
C04197=1087.052,37.065,440.668,174.802,18.914,153.035
C04198=1087.046,36.815,440.683,174.801,18.912,153.035
C04199=1087.040,36.565,440.698,174.799,18.910,153.035
C04200=1087.035,36.316,440.713,174.797,18.908,153.035
C04201=1087.029,36.067,440.729,174.795,18.906,153.035
C04202=1087.023,35.817,440.744,174.794,18.904,153.035
C04203=1087.017,35.568,440.759,174.792,18.903,153.035
C04204=1087.011,35.318,440.775,174.790,18.901,153.035
C04205=1087.006,35.068,440.790,174.789,18.899,153.035
C04206=1087.000,34.819,440.805,174.787,18.897,153.035
C04207=1086.994,34.569,440.821,174.785,18.895,153.035
C04208=1086.988,34.321,440.836,174.784,18.894,153.035
C04209=1086.983,34.071,440.851,174.781,18.892,153.035
C04210=1086.976,33.821,440.866,174.780,18.890,153.034
C04211=1086.971,33.572,440.881,174.779,18.888,153.034
C04212=1086.966,33.322,440.897,174.777,18.886,153.034
C04213=1086.959,33.073,440.912,174.775,18.884,153.034
C04214=1086.954,32.823,440.928,174.774,18.882,153.034
C04215=1086.948,32.574,440.942,174.772,18.880,153.034
C04216=1086.942,32.324,440.958,174.770,18.879,153.034
C04217=1086.936,32.075,440.973,174.768,18.876,153.034
C04218=1086.931,31.825,440.988,174.767,18.875,153.034
C04219=1086.922,31.451,441.010,174.765,18.872,153.034
C04220=1086.914,31.077,441.033,174.762,18.869,153.034
C04221=1086.905,30.702,441.056,174.759,18.866,153.034
C04222=1086.896,30.328,441.079,174.757,18.863,153.033
C04223=1086.890,30.078,441.094,174.756,18.862,153.033
C04224=1086.885,29.829,441.109,174.753,18.860,153.033
C04225=1086.879,29.579,441.124,174.752,18.858,153.033
C04226=1086.873,29.330,441.139,174.750,18.856,153.033
C04227=1086.868,29.080,441.154,174.748,18.854,153.033
C04228=1086.862,28.831,441.169,174.747,18.852,153.033
C04229=1086.856,28.581,441.184,174.745,18.850,153.033
C04230=1086.850,28.332,441.199,174.743,18.849,153.033
C04231=1086.845,28.082,441.215,174.742,18.847,153.033
C04232=1086.839,27.833,441.229,174.740,18.844,153.033
C04233=1086.833,27.584,441.244,174.739,18.843,153.033
C04234=1086.828,27.334,441.259,174.737,18.841,153.033
C04235=1086.821,27.084,441.274,174.735,18.839,153.032
C04236=1086.816,26.835,441.289,174.734,18.837,153.032
C04237=1086.810,26.585,441.304,174.732,18.836,153.032
C04238=1086.804,26.336,441.318,174.730,18.833,153.032
C04239=1086.799,26.086,441.334,174.729,18.832,153.032
C04240=1086.793,25.837,441.348,174.727,18.830,153.032
C04241=1086.786,25.588,441.363,174.725,18.828,153.032
C04242=1086.781,25.338,441.378,174.724,18.826,153.032
C04243=1086.775,25.088,441.393,174.723,18.825,153.032
C04244=1086.770,24.839,441.407,174.720,18.822,153.032
C04245=1086.764,24.589,441.423,174.719,18.820,153.032
C04246=1086.758,24.340,441.437,174.718,18.819,153.032
C04247=1086.752,24.091,441.452,174.715,18.817,153.032
C04248=1086.747,23.841,441.468,174.714,18.815,153.031
C04249=1086.741,23.591,441.482,174.713,18.813,153.031
C04250=1086.735,23.342,441.496,174.710,18.811,153.031
C04251=1086.729,23.092,441.512,174.709,18.809,153.031
C04252=1086.723,22.843,441.526,174.708,18.808,153.031
C04253=1086.717,22.594,441.541,174.706,18.806,153.031
C04254=1086.712,22.344,441.555,174.704,18.804,153.031
C04255=1086.707,22.095,441.570,174.703,18.802,153.031
C04256=1086.700,21.845,441.585,174.701,18.800,153.031
C04257=1086.694,21.596,441.600,174.700,18.798,153.031
C04258=1086.689,21.346,441.615,174.698,18.796,153.031
C04259=1086.683,21.097,441.629,174.696,18.794,153.031
C04260=1086.677,20.847,441.644,174.695,18.792,153.031
C04261=1086.671,20.598,441.659,174.693,18.791,153.030
C04262=1086.666,20.348,441.673,174.691,18.789,153.030
C04263=1086.656,19.946,441.697,174.688,18.786,153.030
C04264=1086.647,19.543,441.721,174.686,18.783,153.030
C04265=1086.638,19.141,441.744,174.683,18.779,153.030
C04266=1086.628,18.738,441.767,174.681,18.776,153.030
C04267=1086.623,18.489,441.783,174.679,18.775,153.030
C04268=1086.617,18.240,441.798,174.678,18.773,153.030
C04269=1086.611,17.990,441.811,174.676,18.771,153.030
C04270=1086.605,17.740,441.826,174.674,18.769,153.030
C04271=1086.599,17.491,441.840,174.673,18.768,153.030
C04272=1086.594,17.242,441.855,174.671,18.765,153.029
C04273=1086.588,16.992,441.870,174.669,18.764,153.029
C04274=1086.583,16.742,441.884,174.668,18.761,153.029
C04275=1086.576,16.493,441.899,174.666,18.759,153.029
C04276=1086.571,16.243,441.913,174.665,18.758,153.029
C04277=1086.565,15.994,441.928,174.663,18.756,153.029
C04278=1086.558,15.744,441.943,174.661,18.754,153.029
C04279=1086.552,15.468,441.958,174.660,18.752,153.029
C04280=1086.546,15.192,441.975,174.658,18.750,153.029
C04281=1086.539,14.915,441.990,174.656,18.748,153.029
C04282=1086.534,14.638,442.006,174.654,18.746,153.029
C04283=1086.528,14.389,442.021,174.653,18.744,153.029
C04284=1086.522,14.140,442.036,174.652,18.742,153.028
C04285=1086.516,13.890,442.050,174.649,18.740,153.028
C04286=1086.510,13.641,442.064,174.648,18.738,153.028
C04287=1086.505,13.391,442.078,174.646,18.737,153.028
C04288=1086.498,13.141,442.093,174.644,18.734,153.028
C04289=1086.492,12.892,442.106,174.643,18.733,153.028
C04290=1086.486,12.643,442.121,174.642,18.731,153.028
C04291=1086.480,12.393,442.135,174.640,18.729,153.028
C04292=1086.475,12.143,442.149,174.638,18.727,153.028
C04293=1086.468,11.894,442.164,174.637,18.726,153.028
C04294=1086.463,11.644,442.178,174.636,18.724,153.028
C04295=1086.457,11.395,442.193,174.633,18.721,153.028
C04296=1086.451,11.145,442.207,174.632,18.720,153.028
C04297=1086.445,10.896,442.221,174.630,18.718,153.028
C04298=1086.440,10.646,442.235,174.628,18.716,153.027
C04299=1086.434,10.396,442.249,174.627,18.714,153.027
C04300=1086.428,10.147,442.264,174.626,18.713,153.027
C04301=1086.422,9.897,442.278,174.624,18.711,153.027
C04302=1086.416,9.648,442.293,174.622,18.709,153.027
C04303=1086.410,9.399,442.306,174.621,18.707,153.027
C04304=1086.404,9.149,442.320,174.619,18.705,153.027
C04305=1086.399,8.900,442.335,174.617,18.703,153.027
C04306=1086.393,8.650,442.349,174.616,18.701,153.027
C04307=1086.387,8.400,442.363,174.615,18.699,153.027
C04308=1086.381,8.151,442.377,174.612,18.697,153.027
C04309=1086.375,7.901,442.391,174.611,18.696,153.027
C04310=1086.370,7.651,442.405,174.610,18.694,153.026
C04311=1086.364,7.402,442.420,174.608,18.692,153.026
C04312=1086.358,7.153,442.433,174.606,18.690,153.026
C04313=1086.352,6.903,442.447,174.605,18.688,153.026
C04314=1086.346,6.654,442.462,174.603,18.687,153.026
C04315=1086.340,6.404,442.476,174.601,18.685,153.026
C04316=1086.335,6.155,442.490,174.600,18.682,153.026
C04317=1086.329,5.904,442.504,174.599,18.681,153.026
C04318=1086.323,5.656,442.519,174.597,18.679,153.026
C04319=1086.318,5.406,442.532,174.595,18.677,153.026
C04320=1086.311,5.157,442.546,174.594,18.675,153.026
C04321=1086.305,4.906,442.560,174.593,18.673,153.026
C04322=1086.299,4.657,442.574,174.591,18.672,153.025
C04323=1086.294,4.408,442.588,174.589,18.670,153.025
C04324=1086.289,4.158,442.602,174.588,18.668,153.025
C04325=1086.282,3.908,442.616,174.586,18.666,153.025
C04326=1086.276,3.659,442.630,174.584,18.664,153.025
C04327=1086.270,3.410,442.644,174.583,18.662,153.025
C04328=1086.265,3.160,442.658,174.581,18.660,153.025
C04329=1086.259,2.911,442.672,174.580,18.659,153.025
C04330=1086.253,2.660,442.686,174.578,18.656,153.025
C04331=1086.248,2.411,442.700,174.576,18.655,153.025
C04332=1086.241,2.162,442.714,174.575,18.653,153.025
C04333=1086.236,1.913,442.728,174.573,18.651,153.025
C04334=1086.230,1.663,442.742,174.572,18.649,153.025
C04335=1086.225,1.413,442.756,174.570,18.647,153.024
C04336=1086.219,1.163,442.770,174.569,18.645,153.024
C04337=1086.213,0.914,442.783,174.567,18.643,153.024
C04338=1086.207,0.664,442.797,174.566,18.641,153.024
C04339=1086.202,0.415,442.811,174.564,18.640,153.024
C04340=1086.196,0.165,442.825,174.563,18.638,153.024
C04341=1086.190,-0.084,442.839,174.561,18.636,153.024
C04342=1086.184,-0.333,442.853,174.559,18.634,153.024
C04343=1086.178,-0.608,442.867,174.558,18.632,153.024
C04344=1086.171,-0.882,442.883,174.556,18.630,153.024
C04345=1086.166,-1.157,442.898,174.555,18.628,153.024
C04346=1086.159,-1.431,442.913,174.553,18.625,153.023
C04347=1086.153,-1.681,442.927,174.551,18.624,153.023
C04348=1086.148,-1.930,442.941,174.550,18.622,153.023
C04349=1086.143,-2.180,442.955,174.548,18.620,153.023
C04350=1086.136,-2.430,442.968,174.546,18.618,153.023
C04351=1086.130,-2.679,442.982,174.545,18.616,153.023
C04352=1086.125,-2.929,442.996,174.544,18.615,153.023
C04353=1086.119,-3.179,443.010,174.542,18.613,153.023
C04354=1086.113,-3.428,443.023,174.540,18.610,153.023
C04355=1086.108,-3.677,443.037,174.539,18.609,153.023
C04356=1086.101,-3.927,443.050,174.537,18.607,153.023
C04357=1086.096,-4.176,443.064,174.536,18.605,153.022
C04358=1086.089,-4.426,443.078,174.534,18.603,153.022
C04359=1086.084,-4.676,443.092,174.533,18.602,153.022
C04360=1086.078,-4.925,443.106,174.531,18.600,153.022
C04361=1086.072,-5.175,443.119,174.529,18.598,153.022
C04362=1086.066,-5.424,443.133,174.528,18.596,153.022
C04363=1086.060,-5.674,443.146,174.526,18.595,153.022
C04364=1086.055,-5.923,443.160,174.525,18.592,153.022
C04365=1086.049,-6.172,443.173,174.523,18.590,153.022
C04366=1086.043,-6.423,443.187,174.522,18.589,153.022
C04367=1086.037,-6.673,443.200,174.520,18.587,153.022
C04368=1086.031,-6.922,443.214,174.519,18.585,153.022
C04369=1086.025,-7.171,443.227,174.517,18.583,153.022
C04370=1086.019,-7.421,443.241,174.516,18.581,153.021
C04371=1086.013,-7.670,443.254,174.514,18.580,153.021
C04372=1086.008,-7.920,443.268,174.513,18.578,153.021
C04373=1086.001,-8.169,443.281,174.510,18.576,153.021
C04374=1085.996,-8.419,443.294,174.509,18.574,153.021
C04375=1085.990,-8.668,443.308,174.508,18.572,153.021
C04376=1085.984,-8.919,443.322,174.506,18.571,153.021
C04377=1085.978,-9.168,443.335,174.504,18.568,153.021
C04378=1085.972,-9.418,443.349,174.503,18.567,153.021
C04379=1085.966,-9.667,443.362,174.502,18.565,153.021
C04380=1085.961,-9.917,443.376,174.500,18.563,153.021
C04381=1085.955,-10.166,443.389,174.498,18.561,153.021
C04382=1085.949,-10.416,443.403,174.497,18.559,153.021
C04383=1085.943,-10.665,443.416,174.496,18.557,153.020
C04384=1085.937,-10.915,443.428,174.494,18.556,153.020
C04385=1085.932,-11.165,443.442,174.493,18.554,153.020
C04386=1085.925,-11.414,443.456,174.491,18.552,153.020
C04387=1085.920,-11.663,443.469,174.489,18.550,153.020
C04388=1085.914,-11.913,443.482,174.488,18.549,153.020
C04389=1085.909,-12.163,443.496,174.487,18.547,153.020
C04390=1085.902,-12.412,443.509,174.484,18.545,153.020
C04391=1085.897,-12.662,443.522,174.483,18.543,153.020
C04392=1085.891,-12.912,443.536,174.482,18.541,153.020
C04393=1085.885,-13.161,443.549,174.480,18.539,153.020
C04394=1085.879,-13.410,443.563,174.478,18.537,153.020
C04395=1085.873,-13.660,443.575,174.477,18.535,153.020
C04396=1085.868,-13.910,443.589,174.476,18.534,153.020
C04397=1085.862,-14.159,443.602,174.474,18.532,153.019
C04398=1085.857,-14.409,443.616,174.473,18.530,153.019
C04399=1085.850,-14.659,443.629,174.471,18.528,153.019
C04400=1085.844,-14.908,443.642,174.469,18.527,153.019
C04401=1085.839,-15.158,443.655,174.468,18.524,153.019
C04402=1085.833,-15.407,443.668,174.467,18.523,153.019
C04403=1085.827,-15.657,443.681,174.464,18.521,153.019
C04404=1085.821,-15.907,443.694,174.463,18.519,153.019
C04405=1085.815,-16.156,443.708,174.462,18.517,153.019
C04406=1085.809,-16.406,443.721,174.460,18.516,153.019
C04407=1085.803,-16.679,443.735,174.458,18.514,153.019
C04408=1085.797,-16.951,443.749,174.457,18.512,153.019
C04409=1085.790,-17.224,443.765,174.456,18.510,153.019
C04410=1085.784,-17.497,443.779,174.453,18.508,153.019
C04411=1085.778,-17.747,443.791,174.452,18.506,153.018
C04412=1085.771,-17.996,443.805,174.451,18.504,153.018
C04413=1085.766,-18.246,443.817,174.449,18.503,153.018
C04414=1085.759,-18.495,443.830,174.447,18.501,153.018
C04415=1085.754,-18.745,443.844,174.446,18.499,153.018
C04416=1085.748,-18.995,443.857,174.444,18.497,153.018
C04417=1085.742,-19.244,443.869,174.443,18.496,153.018
C04418=1085.736,-19.494,443.883,174.442,18.494,153.018
C04419=1085.731,-19.744,443.896,174.440,18.491,153.018
C04420=1085.724,-19.993,443.909,174.438,18.490,153.018
C04421=1085.719,-20.243,443.922,174.437,18.488,153.018
C04422=1085.713,-20.492,443.935,174.435,18.487,153.018
C04423=1085.707,-20.741,443.947,174.434,18.485,153.018
C04424=1085.701,-20.991,443.960,174.432,18.483,153.018
C04425=1085.696,-21.241,443.974,174.430,18.481,153.017
C04426=1085.689,-21.490,443.987,174.429,18.479,153.017
C04427=1085.683,-21.740,443.999,174.428,18.478,153.017
C04428=1085.677,-21.989,444.013,174.426,18.476,153.017
C04429=1085.671,-22.239,444.025,174.424,18.474,153.017
C04430=1085.666,-22.489,444.039,174.423,18.472,153.017
C04431=1085.660,-22.739,444.052,174.422,18.470,153.017
C04432=1085.654,-22.989,444.064,174.420,18.469,153.017
C04433=1085.648,-23.237,444.077,174.419,18.467,153.017
C04434=1085.643,-23.487,444.090,174.417,18.465,153.017
C04435=1085.636,-23.736,444.103,174.415,18.463,153.017
C04436=1085.631,-23.986,444.116,174.414,18.462,153.017
C04437=1085.625,-24.236,444.129,174.413,18.460,153.017
C04438=1085.619,-24.486,444.142,174.411,18.458,153.016
C04439=1085.613,-24.735,444.154,174.409,18.456,153.016
C04440=1085.607,-24.985,444.167,174.408,18.454,153.016
C04441=1085.602,-25.234,444.180,174.406,18.453,153.016
C04442=1085.596,-25.484,444.192,174.405,18.451,153.016
C04443=1085.591,-25.734,444.206,174.404,18.449,153.016
C04444=1085.584,-25.983,444.219,174.402,18.448,153.016
C04445=1085.578,-26.233,444.231,174.400,18.446,153.016
C04446=1085.573,-26.483,444.244,174.399,18.443,153.016
C04447=1085.567,-26.732,444.257,174.397,18.442,153.016
C04448=1085.561,-26.981,444.269,174.396,18.440,153.016
C04449=1085.555,-27.231,444.282,174.395,18.439,153.016
C04450=1085.549,-27.481,444.295,174.393,18.436,153.016
C04451=1085.543,-27.730,444.308,174.391,18.435,153.016
C04452=1085.537,-27.980,444.320,174.390,18.433,153.016
C04453=1085.531,-28.230,444.333,174.388,18.432,153.016
C04454=1085.526,-28.479,444.346,174.387,18.430,153.016
C04455=1085.520,-28.729,444.358,174.385,18.428,153.015
C04456=1085.514,-28.979,444.371,174.383,18.426,153.015
C04457=1085.508,-29.228,444.383,174.382,18.424,153.015
C04458=1085.502,-29.478,444.397,174.381,18.423,153.015
C04459=1085.496,-29.728,444.409,174.379,18.421,153.015
C04460=1085.489,-29.977,444.421,174.378,18.420,153.015
C04461=1085.484,-30.226,444.433,174.376,18.418,153.015
C04462=1085.478,-30.476,444.446,174.374,18.416,153.015
C04463=1085.472,-30.726,444.459,174.373,18.414,153.015
C04464=1085.466,-30.975,444.472,174.372,18.412,153.015
C04465=1085.460,-31.225,444.484,174.370,18.411,153.015
C04466=1085.454,-31.474,444.497,174.369,18.409,153.015
C04467=1085.449,-31.724,444.509,174.368,18.407,153.015
C04468=1085.443,-31.974,444.522,174.365,18.405,153.015
C04469=1085.436,-32.223,444.535,174.364,18.404,153.015
C04470=1085.431,-32.473,444.547,174.362,18.402,153.015
C04471=1085.424,-32.745,444.561,174.361,18.401,153.015
C04472=1085.418,-33.017,444.574,174.359,18.398,153.014
C04473=1085.411,-33.289,444.588,174.358,18.396,153.014
C04474=1085.405,-33.561,444.602,174.356,18.395,153.014
C04475=1085.399,-33.811,444.614,174.355,18.393,153.014
C04476=1085.393,-34.060,444.626,174.353,18.391,153.014
C04477=1085.387,-34.310,444.639,174.351,18.389,153.014
C04478=1085.382,-34.560,444.651,174.350,18.388,153.014
C04479=1085.376,-34.809,444.663,174.349,18.386,153.014
C04480=1085.370,-35.059,444.676,174.347,18.385,153.014
C04481=1085.364,-35.309,444.689,174.346,18.383,153.014
C04482=1085.358,-35.558,444.701,174.344,18.381,153.014
C04483=1085.352,-35.807,444.713,174.342,18.379,153.014
C04484=1085.346,-36.057,444.726,174.341,18.377,153.014
C04485=1085.340,-36.306,444.738,174.339,18.376,153.014
C04486=1085.335,-36.556,444.751,174.338,18.374,153.014
C04487=1085.329,-36.806,444.763,174.337,18.373,153.014
C04488=1085.323,-37.056,444.776,174.335,18.371,153.014
C04489=1085.317,-37.305,444.788,174.334,18.370,153.014
C04490=1085.311,-37.555,444.800,174.332,18.367,153.013
C04491=1085.305,-37.805,444.812,174.330,18.365,153.013
C04492=1085.300,-38.054,444.825,174.329,18.364,153.013
C04493=1085.294,-38.304,444.837,174.328,18.362,153.013
C04494=1085.288,-38.554,444.850,174.326,18.361,153.013
C04495=1085.282,-38.802,444.861,174.325,18.359,153.013
C04496=1085.276,-39.052,444.874,174.323,18.358,153.013
C04497=1085.270,-39.302,444.886,174.321,18.356,153.013
C04498=1085.264,-39.552,444.898,174.320,18.353,153.013
C04499=1085.258,-39.802,444.910,174.318,18.352,153.013
C04500=1085.252,-40.051,444.922,174.317,18.350,153.013
C04501=1085.246,-40.301,444.934,174.316,18.349,153.013
C04502=1085.240,-40.551,444.947,174.314,18.347,153.013
C04503=1085.234,-40.800,444.959,174.313,18.346,153.013
C04504=1085.228,-41.050,444.971,174.311,18.344,153.013
C04505=1085.222,-41.300,444.984,174.309,18.342,153.013
C04506=1085.217,-41.549,444.996,174.308,18.341,153.013
C04507=1085.210,-41.798,445.008,174.306,18.339,153.013
C04508=1085.204,-42.048,445.020,174.305,18.337,153.013
C04509=1085.198,-42.299,445.032,174.303,18.336,153.013
C04510=1085.192,-42.548,445.044,174.302,18.334,153.013
C04511=1085.186,-42.797,445.056,174.301,18.333,153.013
C04512=1085.181,-43.047,445.069,174.299,18.331,153.013
C04513=1085.175,-43.296,445.081,174.297,18.329,153.013
C04514=1085.169,-43.546,445.093,174.296,18.328,153.013
C04515=1085.162,-43.796,445.104,174.294,18.326,153.012
C04516=1085.157,-44.045,445.116,174.293,18.324,153.012
C04517=1085.151,-44.295,445.129,174.292,18.322,153.012
C04518=1085.144,-44.545,445.141,174.290,18.321,153.012
C04519=1085.139,-44.794,445.153,174.289,18.319,153.012
C04520=1085.133,-45.044,445.166,174.287,18.318,153.012
C04521=1085.127,-45.293,445.177,174.286,18.316,153.012
C04522=1085.122,-45.543,445.189,174.284,18.314,153.012
C04523=1085.115,-45.793,445.201,174.282,18.313,153.012
C04524=1085.110,-46.042,445.213,174.281,18.311,153.012
C04525=1085.104,-46.293,445.225,174.279,18.309,153.012
C04526=1085.097,-46.542,445.237,174.278,18.308,153.012
C04527=1085.092,-46.791,445.249,174.277,18.306,153.012
C04528=1085.085,-47.041,445.261,174.275,18.305,153.012
C04529=1085.080,-47.291,445.273,174.274,18.303,153.012
C04530=1085.074,-47.540,445.285,174.272,18.302,153.012
C04531=1085.068,-47.790,445.297,174.270,18.300,153.012
C04532=1085.063,-48.040,445.309,174.269,18.298,153.012
C04533=1085.056,-48.290,445.321,174.267,18.297,153.012
C04534=1085.051,-48.539,445.333,174.266,18.295,153.012
C04535=1085.044,-48.812,445.346,174.264,18.293,153.012
C04536=1085.038,-49.083,445.359,174.263,18.292,153.012
C04537=1085.031,-49.356,445.372,174.261,18.289,153.011
C04538=1085.025,-49.629,445.385,174.260,18.288,153.011
C04539=1085.019,-49.878,445.397,174.258,18.286,153.011
C04540=1085.013,-50.127,445.409,174.257,18.285,153.011
C04541=1085.007,-50.378,445.420,174.255,18.283,153.011
C04542=1085.002,-50.627,445.432,174.254,18.282,153.011
C04543=1084.995,-50.876,445.444,174.253,18.280,153.011
C04544=1084.989,-51.127,445.455,174.251,18.279,153.011
C04545=1084.983,-51.376,445.468,174.249,18.277,153.011
C04546=1084.977,-51.626,445.479,174.247,18.275,153.011
C04547=1084.971,-51.875,445.490,174.246,18.274,153.011
C04548=1084.965,-52.125,445.503,174.244,18.272,153.011
C04549=1084.959,-52.375,445.514,174.243,18.271,153.011
C04550=1084.953,-52.624,445.526,174.242,18.269,153.011
C04551=1084.946,-52.874,445.537,174.240,18.268,153.011
C04552=1084.941,-53.124,445.550,174.238,18.266,153.011
C04553=1084.934,-53.373,445.561,174.237,18.265,153.011
C04554=1084.928,-53.623,445.572,174.236,18.263,153.011
C04555=1084.923,-53.872,445.585,174.234,18.262,153.011
C04556=1084.916,-54.122,445.596,174.233,18.260,153.011
C04557=1084.910,-54.372,445.608,174.231,18.259,153.011
C04558=1084.904,-54.621,445.619,174.229,18.257,153.011
C04559=1084.898,-54.871,445.631,174.227,18.256,153.011
C04560=1084.892,-55.121,445.642,174.226,18.254,153.011
C04561=1084.886,-55.370,445.654,174.225,18.252,153.011
C04562=1084.881,-55.620,445.666,174.223,18.251,153.011
C04563=1084.874,-55.870,445.678,174.222,18.249,153.011
C04564=1084.868,-56.120,445.689,174.220,18.248,153.011
C04565=1084.862,-56.369,445.700,174.219,18.246,153.011
C04566=1084.856,-56.619,445.712,174.217,18.245,153.011
C04567=1084.850,-56.868,445.724,174.216,18.244,153.011
C04568=1084.844,-57.118,445.735,174.215,18.242,153.011
C04569=1084.838,-57.367,445.747,174.213,18.241,153.011
C04570=1084.832,-57.618,445.758,174.212,18.239,153.011
C04571=1084.826,-57.866,445.770,174.210,18.237,153.011
C04572=1084.820,-58.117,445.781,174.209,18.236,153.011
C04573=1084.814,-58.366,445.792,174.207,18.235,153.011
C04574=1084.808,-58.616,445.805,174.206,18.233,153.011
C04575=1084.802,-58.866,445.816,174.204,18.231,153.011
C04576=1084.796,-59.115,445.828,174.202,18.230,153.011
C04577=1084.790,-59.365,445.838,174.201,18.228,153.011
C04578=1084.784,-59.615,445.850,174.199,18.227,153.011
C04579=1084.778,-59.864,445.862,174.198,18.226,153.011
C04580=1084.772,-60.114,445.873,174.196,18.224,153.011
C04581=1084.766,-60.363,445.885,174.195,18.222,153.011
C04582=1084.760,-60.613,445.896,174.193,18.221,153.011
C04583=1084.754,-60.863,445.907,174.192,18.219,153.011
C04584=1084.748,-61.113,445.919,174.190,18.218,153.011
C04585=1084.742,-61.362,445.930,174.189,18.217,153.011
C04586=1084.736,-61.612,445.942,174.187,18.215,153.011
C04587=1084.730,-61.861,445.953,174.186,18.214,153.011
C04588=1084.723,-62.111,445.964,174.185,18.212,153.011
C04589=1084.718,-62.361,445.976,174.183,18.211,153.011
C04590=1084.712,-62.610,445.987,174.182,18.209,153.011
C04591=1084.706,-62.860,445.999,174.180,18.208,153.011
C04592=1084.700,-63.110,446.010,174.179,18.206,153.011
C04593=1084.694,-63.359,446.021,174.177,18.205,153.011
C04594=1084.689,-63.609,446.033,174.176,18.204,153.011
C04595=1084.682,-63.859,446.044,174.174,18.202,153.011
C04596=1084.677,-64.109,446.055,174.173,18.201,153.011
C04597=1084.671,-64.358,446.067,174.171,18.199,153.011
C04598=1084.664,-64.608,446.078,174.170,18.198,153.011
C04599=1084.658,-64.881,446.090,174.168,18.196,153.011
C04600=1084.652,-65.155,446.102,174.166,18.194,153.011
C04601=1084.645,-65.429,446.115,174.165,18.193,153.011
C04602=1084.638,-65.703,446.127,174.163,18.191,153.011
C04603=1084.632,-65.952,446.139,174.162,18.190,153.011
C04604=1084.627,-66.201,446.150,174.160,18.188,153.011
C04605=1084.620,-66.451,446.161,174.159,18.187,153.011
C04606=1084.615,-66.701,446.172,174.157,18.186,153.011
C04607=1084.609,-66.951,446.184,174.156,18.184,153.011
C04608=1084.603,-67.200,446.195,174.155,18.182,153.011
C04609=1084.597,-67.450,446.206,174.153,18.181,153.011
C04610=1084.591,-67.700,446.217,174.151,18.179,153.011
C04611=1084.585,-67.950,446.228,174.149,18.178,153.011
C04612=1084.579,-68.199,446.239,174.148,18.176,153.011
C04613=1084.573,-68.449,446.250,174.146,18.175,153.011
C04614=1084.567,-68.698,446.262,174.145,18.174,153.011
C04615=1084.562,-68.948,446.273,174.143,18.172,153.011
C04616=1084.556,-69.198,446.285,174.142,18.171,153.011
C04617=1084.550,-69.448,446.296,174.140,18.169,153.011
C04618=1084.544,-69.697,446.306,174.139,18.168,153.011
C04619=1084.538,-69.947,446.318,174.137,18.166,153.011
C04620=1084.532,-70.197,446.329,174.136,18.165,153.011
C04621=1084.526,-70.446,446.339,174.134,18.164,153.011
C04622=1084.520,-70.696,446.351,174.133,18.162,153.011
C04623=1084.514,-70.945,446.362,174.132,18.161,153.011
C04624=1084.508,-71.195,446.373,174.130,18.160,153.011
C04625=1084.503,-71.445,446.385,174.128,18.158,153.011
C04626=1084.497,-71.695,446.396,174.127,18.156,153.011
C04627=1084.491,-71.944,446.407,174.126,18.155,153.011
C04628=1084.485,-72.194,446.418,174.124,18.154,153.011
C04629=1084.479,-72.444,446.429,174.123,18.152,153.011
C04630=1084.473,-72.693,446.440,174.121,18.151,153.011
C04631=1084.468,-72.943,446.451,174.119,18.150,153.011
C04632=1084.461,-73.193,446.462,174.118,18.148,153.011
C04633=1084.455,-73.443,446.473,174.117,18.147,153.011
C04634=1084.450,-73.692,446.484,174.115,18.146,153.011
C04635=1084.444,-73.942,446.494,174.114,18.144,153.011
C04636=1084.438,-74.192,446.506,174.112,18.142,153.011
C04637=1084.432,-74.441,446.517,174.110,18.141,153.011
C04638=1084.426,-74.691,446.527,174.109,18.140,153.011
C04639=1084.420,-74.941,446.539,174.108,18.138,153.011
C04640=1084.414,-75.190,446.550,174.107,18.138,153.011
C04641=1084.408,-75.440,446.560,174.105,18.136,153.011
C04642=1084.401,-75.690,446.571,174.104,18.135,153.011
C04643=1084.396,-75.939,446.582,174.102,18.134,153.011
C04644=1084.390,-76.189,446.593,174.101,18.133,153.011
C04645=1084.384,-76.438,446.604,174.099,18.131,153.011
C04646=1084.378,-76.688,446.615,174.098,18.129,153.011
C04647=1084.372,-76.938,446.626,174.096,18.128,153.011
C04648=1084.366,-77.187,446.637,174.095,18.127,153.011
C04649=1084.359,-77.437,446.647,174.093,18.126,153.011
C04650=1084.354,-77.687,446.658,174.092,18.124,153.011
C04651=1084.348,-77.937,446.668,174.090,18.123,153.011
C04652=1084.342,-78.186,446.679,174.089,18.122,153.011
C04653=1084.336,-78.437,446.691,174.087,18.120,153.011
C04654=1084.330,-78.686,446.701,174.086,18.119,153.011
C04655=1084.324,-78.935,446.712,174.084,18.118,153.011
C04656=1084.318,-79.185,446.723,174.082,18.117,153.011
C04657=1084.312,-79.435,446.734,174.081,18.115,153.011
C04658=1084.306,-79.685,446.744,174.079,18.114,153.012
C04659=1084.300,-79.935,446.755,174.078,18.112,153.012
C04660=1084.294,-80.184,446.765,174.076,18.111,153.012
C04661=1084.288,-80.434,446.776,174.075,18.110,153.012
C04662=1084.282,-80.683,446.787,174.073,18.109,153.012
C04663=1084.275,-80.960,446.799,174.072,18.107,153.012
C04664=1084.268,-81.235,446.811,174.070,18.106,153.012
C04665=1084.262,-81.511,446.822,174.069,18.105,153.012
C04666=1084.254,-81.787,446.834,174.067,18.104,153.012
C04667=1084.249,-82.037,446.845,174.065,18.102,153.012
C04668=1084.242,-82.286,446.855,174.064,18.101,153.012
C04669=1084.236,-82.536,446.866,174.062,18.100,153.012
C04670=1084.230,-82.786,446.877,174.061,18.098,153.012
C04671=1084.224,-83.035,446.887,174.059,18.097,153.012
C04672=1084.218,-83.285,446.897,174.058,18.096,153.012
C04673=1084.212,-83.535,446.909,174.056,18.095,153.012
C04674=1084.206,-83.784,446.919,174.054,18.094,153.012
C04675=1084.200,-84.034,446.930,174.053,18.092,153.012
C04676=1084.194,-84.283,446.939,174.051,18.091,153.012
C04677=1084.187,-84.534,446.951,174.050,18.089,153.012
C04678=1084.182,-84.783,446.962,174.048,18.088,153.012
C04679=1084.175,-85.033,446.971,174.047,18.087,153.013
C04680=1084.170,-85.282,446.982,174.046,18.086,153.013
C04681=1084.164,-85.532,446.993,174.044,18.085,153.013
C04682=1084.157,-85.782,447.003,174.043,18.084,153.013
C04683=1084.151,-86.032,447.014,174.041,18.083,153.013
C04684=1084.145,-86.281,447.024,174.040,18.082,153.013
C04685=1084.139,-86.531,447.035,174.038,18.080,153.013
C04686=1084.134,-86.781,447.045,174.037,18.079,153.013
C04687=1084.127,-87.031,447.056,174.035,18.078,153.013
C04688=1084.121,-87.280,447.066,174.033,18.077,153.013
C04689=1084.115,-87.530,447.076,174.032,18.075,153.013
C04690=1084.109,-87.779,447.087,174.030,18.074,153.013
C04691=1084.103,-88.029,447.097,174.029,18.073,153.013
C04692=1084.097,-88.279,447.108,174.028,18.072,153.013
C04693=1084.091,-88.529,447.119,174.026,18.071,153.013
C04694=1084.084,-88.778,447.129,174.025,18.070,153.013
C04695=1084.079,-89.028,447.139,174.023,18.069,153.013
C04696=1084.072,-89.277,447.149,174.021,18.068,153.014
C04697=1084.067,-89.527,447.160,174.020,18.066,153.014
C04698=1084.060,-89.777,447.170,174.018,18.065,153.014
C04699=1084.054,-90.027,447.181,174.017,18.064,153.014
C04700=1084.049,-90.277,447.191,174.015,18.062,153.014
C04701=1084.042,-90.526,447.201,174.014,18.061,153.014
C04702=1084.037,-90.776,447.212,174.012,18.060,153.014
C04703=1084.030,-91.025,447.222,174.011,18.059,153.014
C04704=1084.025,-91.275,447.232,174.010,18.058,153.014
C04705=1084.018,-91.525,447.242,174.008,18.057,153.014
C04706=1084.012,-91.775,447.254,174.007,18.056,153.014
C04707=1084.006,-92.025,447.263,174.005,18.055,153.014
C04708=1084.000,-92.274,447.274,174.003,18.054,153.014
C04709=1083.994,-92.524,447.284,174.002,18.052,153.014
C04710=1083.988,-92.773,447.295,174.000,18.051,153.014
C04711=1083.983,-93.024,447.305,173.999,18.050,153.014
C04712=1083.976,-93.273,447.315,173.997,18.049,153.015
C04713=1083.971,-93.523,447.325,173.996,18.048,153.014
C04714=1083.964,-93.772,447.335,173.995,18.047,153.015
C04715=1083.959,-94.022,447.346,173.993,18.046,153.015
C04716=1083.952,-94.272,447.356,173.991,18.045,153.015
C04717=1083.947,-94.522,447.366,173.990,18.043,153.015
C04718=1083.940,-94.771,447.377,173.988,18.042,153.015
C04719=1083.935,-95.021,447.387,173.987,18.041,153.015
C04720=1083.928,-95.271,447.397,173.985,18.040,153.015
C04721=1083.923,-95.521,447.407,173.983,18.039,153.015
C04722=1083.917,-95.770,447.417,173.983,18.038,153.015
C04723=1083.911,-96.020,447.428,173.981,18.037,153.015
C04724=1083.905,-96.270,447.437,173.979,18.036,153.015
C04725=1083.899,-96.519,447.448,173.978,18.034,153.015
C04726=1083.893,-96.769,447.458,173.976,18.033,153.015
C04727=1083.886,-97.047,447.469,173.975,18.032,153.016
C04728=1083.879,-97.325,447.480,173.973,18.031,153.016
C04729=1083.873,-97.603,447.492,173.971,18.030,153.016
C04730=1083.866,-97.881,447.503,173.970,18.029,153.016
C04731=1083.860,-98.131,447.513,173.968,18.028,153.016
C04732=1083.854,-98.381,447.523,173.966,18.027,153.016
C04733=1083.847,-98.631,447.533,173.965,18.026,153.016
C04734=1083.842,-98.881,447.543,173.963,18.025,153.016
C04735=1083.835,-99.130,447.554,173.961,18.024,153.016
C04736=1083.829,-99.380,447.563,173.961,18.022,153.016
C04737=1083.824,-99.630,447.573,173.959,18.021,153.016
C04738=1083.817,-99.879,447.584,173.958,18.020,153.016
C04739=1083.811,-100.129,447.593,173.956,18.019,153.017
C04740=1083.805,-100.379,447.603,173.954,18.018,153.017
C04741=1083.799,-100.628,447.614,173.953,18.017,153.017
C04742=1083.793,-100.878,447.623,173.951,18.016,153.017
C04743=1083.787,-101.128,447.633,173.950,18.016,153.017
C04744=1083.781,-101.377,447.644,173.948,18.015,153.017
C04745=1083.775,-101.627,447.653,173.947,18.014,153.017
C04746=1083.769,-101.877,447.663,173.945,18.013,153.017
C04747=1083.762,-102.127,447.672,173.944,18.011,153.017
C04748=1083.757,-102.376,447.683,173.942,18.010,153.017
C04749=1083.751,-102.626,447.693,173.941,18.009,153.018
C04750=1083.744,-102.876,447.702,173.939,18.008,153.018
C04751=1083.738,-103.125,447.713,173.938,18.007,153.018
C04752=1083.732,-103.375,447.723,173.936,18.006,153.018
C04753=1083.726,-103.625,447.733,173.934,18.005,153.018
C04754=1083.719,-103.875,447.742,173.933,18.004,153.018
C04755=1083.713,-104.124,447.753,173.932,18.004,153.018
C04756=1083.708,-104.375,447.763,173.930,18.003,153.018
C04757=1083.701,-104.624,447.772,173.929,18.002,153.018
C04758=1083.695,-104.874,447.782,173.927,18.001,153.018
C04759=1083.690,-105.123,447.791,173.925,18.000,153.019
C04760=1083.684,-105.373,447.802,173.924,17.999,153.019
C04761=1083.678,-105.622,447.812,173.923,17.998,153.019
C04762=1083.672,-105.872,447.821,173.921,17.997,153.019
C04763=1083.665,-106.122,447.831,173.919,17.996,153.019
C04764=1083.659,-106.372,447.840,173.918,17.995,153.019
C04765=1083.653,-106.621,447.851,173.916,17.994,153.019
C04766=1083.647,-106.871,447.861,173.914,17.993,153.019
C04767=1083.641,-107.121,447.870,173.914,17.992,153.019
C04768=1083.635,-107.371,447.880,173.912,17.991,153.020
C04769=1083.629,-107.621,447.889,173.910,17.990,153.020
C04770=1083.623,-107.870,447.899,173.909,17.989,153.020
C04771=1083.617,-108.120,447.910,173.907,17.988,153.020
C04772=1083.611,-108.370,447.919,173.906,17.988,153.020
C04773=1083.605,-108.619,447.929,173.904,17.987,153.020
C04774=1083.598,-108.869,447.939,173.903,17.986,153.020
C04775=1083.592,-109.119,447.948,173.901,17.985,153.020
C04776=1083.586,-109.369,447.958,173.899,17.984,153.021
C04777=1083.580,-109.619,447.967,173.898,17.984,153.021
C04778=1083.574,-109.868,447.977,173.897,17.983,153.021
C04779=1083.567,-110.118,447.987,173.895,17.981,153.021
C04780=1083.561,-110.367,447.997,173.893,17.980,153.021
C04781=1083.555,-110.617,448.006,173.892,17.979,153.021
C04782=1083.549,-110.867,448.016,173.891,17.979,153.021
C04783=1083.543,-111.117,448.026,173.889,17.978,153.021
C04784=1083.537,-111.367,448.036,173.887,17.977,153.022
C04785=1083.531,-111.617,448.045,173.885,17.976,153.022
C04786=1083.525,-111.867,448.055,173.884,17.975,153.022
C04787=1083.519,-112.116,448.064,173.883,17.975,153.022
C04788=1083.513,-112.365,448.074,173.881,17.974,153.022
C04789=1083.507,-112.615,448.083,173.880,17.973,153.022
C04790=1083.501,-112.865,448.093,173.878,17.972,153.022
C04791=1083.494,-113.139,448.104,173.876,17.971,153.022
C04792=1083.487,-113.413,448.114,173.874,17.970,153.023
C04793=1083.481,-113.687,448.125,173.873,17.969,153.023
C04794=1083.474,-113.962,448.134,173.871,17.968,153.023
C04795=1083.467,-114.211,448.144,173.870,17.967,153.023
C04796=1083.462,-114.462,448.154,173.868,17.967,153.023
C04797=1083.455,-114.711,448.163,173.867,17.966,153.023
C04798=1083.449,-114.961,448.173,173.865,17.965,153.023
C04799=1083.443,-115.211,448.182,173.863,17.964,153.023
C04800=1083.437,-115.460,448.192,173.862,17.963,153.024
C04801=1083.430,-115.710,448.201,173.860,17.963,153.024
C04802=1083.425,-115.959,448.210,173.859,17.962,153.024
C04803=1083.419,-116.209,448.220,173.857,17.961,153.024
C04804=1083.412,-116.459,448.230,173.856,17.960,153.024
C04805=1083.406,-116.709,448.239,173.854,17.960,153.024
C04806=1083.400,-116.958,448.249,173.853,17.959,153.024
C04807=1083.394,-117.208,448.258,173.851,17.958,153.025
C04808=1083.388,-117.458,448.268,173.850,17.957,153.025
C04809=1083.382,-117.708,448.277,173.848,17.957,153.025
C04810=1083.375,-117.958,448.287,173.847,17.956,153.025
C04811=1083.370,-118.207,448.295,173.845,17.955,153.025
C04812=1083.364,-118.457,448.305,173.844,17.955,153.025
C04813=1083.357,-118.707,448.314,173.842,17.954,153.025
C04814=1083.351,-118.956,448.324,173.840,17.952,153.026
C04815=1083.345,-119.206,448.333,173.839,17.952,153.026
C04816=1083.339,-119.456,448.343,173.838,17.951,153.026
C04817=1083.332,-119.706,448.352,173.836,17.950,153.026
C04818=1083.326,-119.956,448.362,173.834,17.950,153.026
C04819=1083.321,-120.205,448.370,173.832,17.949,153.026
C04820=1083.315,-120.455,448.380,173.832,17.948,153.026
C04821=1083.309,-120.705,448.389,173.830,17.948,153.027
C04822=1083.302,-120.954,448.398,173.828,17.947,153.027
C04823=1083.296,-121.204,448.408,173.826,17.946,153.027
C04824=1083.289,-121.454,448.418,173.825,17.946,153.027
C04825=1083.284,-121.704,448.426,173.824,17.945,153.027
C04826=1083.278,-121.954,448.436,173.822,17.944,153.027
C04827=1083.272,-122.203,448.445,173.820,17.943,153.028
C04828=1083.265,-122.453,448.454,173.819,17.943,153.028
C04829=1083.259,-122.703,448.464,173.817,17.942,153.028
C04830=1083.253,-122.953,448.473,173.815,17.941,153.028
C04831=1083.247,-123.202,448.482,173.814,17.940,153.028
C04832=1083.241,-123.452,448.491,173.813,17.940,153.028
C04833=1083.235,-123.702,448.501,173.811,17.939,153.029
C04834=1083.228,-123.952,448.509,173.809,17.938,153.029
C04835=1083.222,-124.202,448.519,173.807,17.938,153.029
C04836=1083.217,-124.451,448.528,173.807,17.937,153.029
C04837=1083.210,-124.701,448.537,173.805,17.936,153.029
C04838=1083.205,-124.951,448.546,173.803,17.935,153.029
C04839=1083.198,-125.200,448.555,173.802,17.935,153.030
C04840=1083.191,-125.450,448.565,173.800,17.934,153.030
C04841=1083.185,-125.700,448.574,173.799,17.933,153.030
C04842=1083.179,-125.949,448.582,173.797,17.933,153.030
C04843=1083.173,-126.199,448.592,173.796,17.932,153.030
C04844=1083.167,-126.449,448.601,173.794,17.932,153.030
C04845=1083.161,-126.699,448.610,173.792,17.931,153.031
C04846=1083.154,-126.949,448.619,173.791,17.931,153.031
C04847=1083.149,-127.198,448.628,173.789,17.930,153.031
C04848=1083.142,-127.448,448.638,173.787,17.929,153.031
C04849=1083.136,-127.698,448.646,173.786,17.928,153.031
C04850=1083.130,-127.948,448.656,173.785,17.928,153.031
C04851=1083.125,-128.205,448.665,173.783,17.927,153.032
C04852=1083.124,-128.460,448.676,173.782,17.925,153.031
C04853=1083.128,-128.715,448.689,173.782,17.921,153.031
C04854=1083.136,-128.967,448.703,173.782,17.917,153.030
C04855=1082.735,-128.989,448.567,173.737,18.034,153.060
C04856=1082.727,-128.736,448.553,173.738,18.039,153.061
C04857=1082.724,-128.481,448.541,173.739,18.042,153.061
C04858=1082.724,-128.226,448.530,173.740,18.044,153.062
C04859=1082.728,-127.970,448.519,173.740,18.045,153.062
C04860=1082.735,-127.720,448.510,173.742,18.046,153.061
C04861=1082.740,-127.471,448.502,173.744,18.047,153.061
C04862=1082.747,-127.221,448.492,173.746,18.047,153.061
C04863=1082.754,-126.971,448.483,173.747,18.048,153.061
C04864=1082.759,-126.721,448.474,173.749,18.048,153.061
C04865=1082.766,-126.471,448.465,173.750,18.050,153.061
C04866=1082.771,-126.222,448.456,173.751,18.049,153.060
C04867=1082.778,-125.972,448.447,173.753,18.051,153.060
C04868=1082.784,-125.722,448.438,173.755,18.051,153.060
C04869=1082.790,-125.472,448.428,173.757,18.052,153.060
C04870=1082.797,-125.223,448.419,173.757,18.053,153.060
C04871=1082.803,-124.972,448.410,173.759,18.053,153.060
C04872=1082.808,-124.723,448.401,173.761,18.054,153.059
C04873=1082.815,-124.473,448.392,173.762,18.054,153.059
C04874=1082.822,-124.224,448.383,173.764,18.055,153.059
C04875=1082.827,-123.974,448.374,173.766,18.056,153.059
C04876=1082.834,-123.724,448.364,173.767,18.057,153.059
C04877=1082.839,-123.475,448.355,173.768,18.057,153.059
C04878=1082.845,-123.225,448.346,173.770,18.058,153.058
C04879=1082.851,-122.974,448.337,173.772,18.059,153.058
C04880=1082.858,-122.725,448.328,173.774,18.060,153.058
C04881=1082.864,-122.475,448.318,173.775,18.060,153.058
C04882=1082.870,-122.226,448.309,173.776,18.061,153.058
C04883=1082.876,-121.976,448.299,173.778,18.062,153.058
C04884=1082.882,-121.726,448.291,173.780,18.062,153.058
C04885=1082.888,-121.476,448.281,173.781,18.063,153.057
C04886=1082.895,-121.227,448.272,173.782,18.064,153.057
C04887=1082.901,-120.977,448.262,173.784,18.064,153.057
C04888=1082.907,-120.727,448.253,173.786,18.065,153.057
C04889=1082.913,-120.477,448.244,173.787,18.066,153.057
C04890=1082.919,-120.227,448.235,173.789,18.066,153.057
C04891=1082.925,-119.978,448.225,173.791,18.067,153.057
C04892=1082.931,-119.728,448.216,173.792,18.068,153.056
C04893=1082.937,-119.478,448.206,173.793,18.069,153.056
C04894=1082.944,-119.229,448.197,173.795,18.069,153.056
C04895=1082.950,-118.979,448.188,173.797,18.070,153.056
C04896=1082.956,-118.730,448.178,173.798,18.072,153.056
C04897=1082.962,-118.479,448.170,173.799,18.072,153.056
C04898=1082.968,-118.229,448.160,173.801,18.073,153.055
C04899=1082.974,-117.980,448.150,173.803,18.074,153.055
C04900=1082.980,-117.730,448.141,173.804,18.075,153.055
C04901=1082.986,-117.480,448.131,173.806,18.075,153.055
C04902=1082.993,-117.230,448.122,173.807,18.076,153.055
C04903=1082.999,-116.980,448.112,173.809,18.077,153.055
C04904=1083.004,-116.731,448.103,173.811,18.078,153.055
C04905=1083.011,-116.482,448.093,173.813,18.078,153.054
C04906=1083.017,-116.232,448.084,173.813,18.079,153.054
C04907=1083.024,-115.982,448.075,173.815,18.080,153.054
C04908=1083.030,-115.732,448.065,173.817,18.081,153.054
C04909=1083.036,-115.483,448.056,173.818,18.082,153.054
C04910=1083.042,-115.232,448.047,173.819,18.082,153.054
C04911=1083.048,-114.982,448.037,173.821,18.083,153.054
C04912=1083.054,-114.733,448.028,173.823,18.084,153.054
C04913=1083.060,-114.483,448.018,173.824,18.085,153.053
C04914=1083.066,-114.234,448.009,173.826,18.086,153.053
C04915=1083.072,-113.984,447.999,173.827,18.086,153.053
C04916=1083.079,-113.709,447.988,173.829,18.087,153.053
C04917=1083.086,-113.435,447.978,173.831,18.088,153.053
C04918=1083.093,-113.161,447.967,173.832,18.089,153.053
C04919=1083.099,-112.886,447.957,173.834,18.090,153.053
C04920=1083.105,-112.637,447.947,173.836,18.091,153.053
C04921=1083.111,-112.387,447.938,173.837,18.092,153.052
C04922=1083.118,-112.137,447.928,173.839,18.093,153.052
C04923=1083.124,-111.887,447.918,173.840,18.093,153.052
C04924=1083.130,-111.637,447.909,173.842,18.094,153.052
C04925=1083.136,-111.388,447.899,173.843,18.095,153.052
C04926=1083.142,-111.138,447.890,173.845,18.096,153.052
C04927=1083.148,-110.888,447.880,173.847,18.097,153.052
C04928=1083.154,-110.638,447.870,173.848,18.098,153.052
C04929=1083.159,-110.389,447.861,173.849,18.099,153.051
C04930=1083.166,-110.140,447.851,173.851,18.100,153.051
C04931=1083.172,-109.890,447.841,173.853,18.101,153.051
C04932=1083.178,-109.640,447.831,173.854,18.102,153.051
C04933=1083.184,-109.390,447.822,173.855,18.102,153.051
C04934=1083.191,-109.140,447.812,173.857,18.103,153.051
C04935=1083.197,-108.891,447.803,173.859,18.104,153.051
C04936=1083.203,-108.641,447.793,173.860,18.105,153.051
C04937=1083.209,-108.391,447.784,173.862,18.106,153.050
C04938=1083.215,-108.141,447.774,173.864,18.107,153.050
C04939=1083.221,-107.892,447.763,173.865,18.108,153.050
C04940=1083.227,-107.642,447.754,173.866,18.109,153.050
C04941=1083.233,-107.392,447.744,173.868,18.110,153.050
C04942=1083.239,-107.142,447.734,173.870,18.111,153.050
C04943=1083.246,-106.892,447.725,173.871,18.112,153.050
C04944=1083.252,-106.643,447.715,173.872,18.112,153.050
C04945=1083.258,-106.393,447.704,173.874,18.113,153.050
C04946=1083.264,-106.143,447.695,173.875,18.114,153.050
C04947=1083.270,-105.894,447.685,173.877,18.115,153.049
C04948=1083.276,-105.644,447.676,173.879,18.116,153.049
C04949=1083.282,-105.394,447.666,173.881,18.117,153.049
C04950=1083.288,-105.145,447.655,173.881,18.118,153.049
C04951=1083.294,-104.895,447.646,173.883,18.119,153.049
C04952=1083.300,-104.645,447.636,173.885,18.120,153.049
C04953=1083.307,-104.395,447.627,173.886,18.121,153.049
C04954=1083.312,-104.145,447.616,173.888,18.123,153.049
C04955=1083.318,-103.896,447.606,173.889,18.124,153.049
C04956=1083.325,-103.646,447.597,173.890,18.124,153.049
C04957=1083.331,-103.396,447.587,173.892,18.125,153.049
C04958=1083.336,-103.146,447.577,173.894,18.126,153.048
C04959=1083.343,-102.897,447.567,173.895,18.127,153.048
C04960=1083.349,-102.647,447.557,173.897,18.128,153.048
C04961=1083.355,-102.397,447.547,173.899,18.129,153.048
C04962=1083.361,-102.148,447.537,173.900,18.130,153.048
C04963=1083.367,-101.898,447.527,173.901,18.131,153.048
C04964=1083.373,-101.648,447.517,173.903,18.132,153.048
C04965=1083.379,-101.398,447.508,173.904,18.133,153.048
C04966=1083.385,-101.149,447.497,173.906,18.134,153.048
C04967=1083.391,-100.899,447.487,173.908,18.135,153.048
C04968=1083.397,-100.649,447.478,173.909,18.136,153.047
C04969=1083.403,-100.400,447.467,173.911,18.137,153.047
C04970=1083.409,-100.150,447.457,173.912,18.138,153.047
C04971=1083.415,-99.900,447.448,173.913,18.139,153.047
C04972=1083.423,-99.650,447.437,173.915,18.140,153.047
C04973=1083.428,-99.400,447.427,173.917,18.142,153.047
C04974=1083.434,-99.151,447.417,173.918,18.143,153.047
C04975=1083.441,-98.901,447.407,173.920,18.144,153.047
C04976=1083.446,-98.651,447.397,173.922,18.145,153.047
C04977=1083.453,-98.402,447.387,173.922,18.145,153.047
C04978=1083.459,-98.152,447.377,173.924,18.146,153.047
C04979=1083.464,-97.902,447.367,173.925,18.148,153.047
C04980=1083.471,-97.625,447.356,173.927,18.149,153.046
C04981=1083.478,-97.347,447.344,173.929,18.150,153.046
C04982=1083.485,-97.068,447.333,173.931,18.151,153.046
C04983=1083.492,-96.790,447.321,173.932,18.152,153.046
C04984=1083.497,-96.540,447.311,173.934,18.153,153.046
C04985=1083.503,-96.290,447.302,173.935,18.155,153.046
C04986=1083.509,-96.040,447.291,173.937,18.156,153.046
C04987=1083.515,-95.790,447.281,173.938,18.157,153.046
C04988=1083.521,-95.541,447.270,173.940,18.158,153.046
C04989=1083.527,-95.291,447.261,173.942,18.159,153.046
C04990=1083.533,-95.042,447.250,173.943,18.161,153.046
C04991=1083.539,-94.792,447.240,173.945,18.162,153.046
C04992=1083.545,-94.542,447.230,173.946,18.162,153.046
C04993=1083.551,-94.293,447.220,173.947,18.163,153.045
C04994=1083.557,-94.043,447.209,173.949,18.165,153.045
C04995=1083.563,-93.793,447.200,173.950,18.166,153.045
C04996=1083.569,-93.543,447.188,173.952,18.167,153.045
C04997=1083.575,-93.293,447.179,173.953,18.168,153.045
C04998=1083.581,-93.044,447.168,173.955,18.170,153.045
C04999=1083.587,-92.794,447.158,173.957,18.171,153.045
C05000=1083.593,-92.545,447.147,173.958,18.172,153.045
C05001=1083.599,-92.295,447.138,173.960,18.173,153.045
C05002=1083.605,-92.045,447.127,173.961,18.174,153.045
C05003=1083.611,-91.795,447.117,173.962,18.175,153.045
C05004=1083.617,-91.546,447.107,173.964,18.176,153.045
C05005=1083.624,-91.295,447.097,173.966,18.177,153.045
C05006=1083.629,-91.046,447.086,173.967,18.179,153.045
C05007=1083.635,-90.796,447.076,173.969,18.180,153.045
C05008=1083.641,-90.547,447.065,173.970,18.181,153.045
C05009=1083.647,-90.297,447.054,173.972,18.182,153.045
C05010=1083.653,-90.047,447.045,173.973,18.183,153.044
C05011=1083.659,-89.798,447.034,173.975,18.185,153.044
C05012=1083.666,-89.547,447.024,173.976,18.186,153.044
C05013=1083.671,-89.298,447.013,173.977,18.187,153.044
C05014=1083.678,-89.049,447.003,173.979,18.188,153.044
C05015=1083.683,-88.799,446.993,173.980,18.189,153.044
C05016=1083.689,-88.549,446.982,173.982,18.190,153.044
C05017=1083.695,-88.300,446.972,173.983,18.192,153.044
C05018=1083.702,-88.049,446.961,173.985,18.193,153.044
C05019=1083.708,-87.800,446.951,173.987,18.194,153.044
C05020=1083.713,-87.550,446.941,173.988,18.195,153.044
C05021=1083.719,-87.300,446.930,173.990,18.196,153.044
C05022=1083.726,-87.051,446.919,173.991,18.198,153.044
C05023=1083.731,-86.801,446.909,173.993,18.199,153.044
C05024=1083.738,-86.551,446.899,173.994,18.201,153.044
C05025=1083.744,-86.302,446.888,173.995,18.201,153.044
C05026=1083.750,-86.053,446.877,173.997,18.202,153.044
C05027=1083.756,-85.802,446.867,173.998,18.204,153.044
C05028=1083.762,-85.553,446.856,174.000,18.205,153.044
C05029=1083.769,-85.303,446.846,174.001,18.206,153.044
C05030=1083.774,-85.053,446.836,174.003,18.207,153.043
C05031=1083.780,-84.803,446.825,174.005,18.208,153.043
C05032=1083.786,-84.554,446.814,174.006,18.210,153.043
C05033=1083.793,-84.304,446.803,174.008,18.211,153.043
C05034=1083.799,-84.054,446.794,174.009,18.212,153.043
C05035=1083.805,-83.805,446.783,174.011,18.213,153.043
C05036=1083.810,-83.555,446.772,174.012,18.215,153.043
C05037=1083.817,-83.305,446.761,174.014,18.216,153.043
C05038=1083.823,-83.055,446.751,174.015,18.218,153.043
C05039=1083.829,-82.806,446.740,174.017,18.219,153.043
C05040=1083.835,-82.557,446.730,174.019,18.220,153.043
C05041=1083.841,-82.306,446.719,174.019,18.221,153.043
C05042=1083.847,-82.057,446.708,174.021,18.222,153.043
C05043=1083.853,-81.807,446.698,174.022,18.223,153.043
C05044=1083.860,-81.532,446.686,174.024,18.224,153.043
C05045=1083.867,-81.255,446.674,174.026,18.226,153.043
C05046=1083.873,-80.979,446.662,174.028,18.227,153.043
C05047=1083.880,-80.704,446.650,174.029,18.229,153.043
C05048=1083.887,-80.454,446.640,174.031,18.230,153.043
C05049=1083.893,-80.204,446.630,174.033,18.232,153.043
C05050=1083.898,-79.954,446.619,174.034,18.233,153.043
C05051=1083.904,-79.705,446.608,174.036,18.234,153.043
C05052=1083.911,-79.455,446.597,174.037,18.236,153.043
C05053=1083.917,-79.205,446.586,174.039,18.237,153.042
C05054=1083.923,-78.956,446.575,174.040,18.238,153.043
C05055=1083.928,-78.706,446.565,174.042,18.239,153.042
C05056=1083.935,-78.456,446.553,174.043,18.241,153.042
C05057=1083.940,-78.206,446.543,174.045,18.242,153.042
C05058=1083.947,-77.957,446.533,174.046,18.243,153.042
C05059=1083.953,-77.707,446.522,174.048,18.245,153.042
C05060=1083.959,-77.457,446.511,174.049,18.246,153.042
C05061=1083.964,-77.208,446.500,174.050,18.247,153.042
C05062=1083.970,-76.958,446.489,174.052,18.248,153.042
C05063=1083.977,-76.708,446.478,174.053,18.250,153.042
C05064=1083.983,-76.459,446.467,174.055,18.251,153.042
C05065=1083.989,-76.209,446.457,174.056,18.252,153.042
C05066=1083.995,-75.959,446.445,174.058,18.254,153.042
C05067=1084.001,-75.710,446.434,174.059,18.255,153.042
C05068=1084.007,-75.460,446.424,174.061,18.256,153.042
C05069=1084.012,-75.211,446.413,174.062,18.258,153.042
C05070=1084.019,-74.961,446.401,174.064,18.259,153.042
C05071=1084.024,-74.711,446.391,174.065,18.261,153.042
C05072=1084.031,-74.462,446.380,174.067,18.262,153.042
C05073=1084.037,-74.212,446.369,174.068,18.263,153.042
C05074=1084.043,-73.962,446.358,174.070,18.265,153.042
C05075=1084.049,-73.713,446.347,174.071,18.266,153.042
C05076=1084.055,-73.462,446.336,174.073,18.268,153.042
C05077=1084.061,-73.213,446.325,174.074,18.269,153.042
C05078=1084.066,-72.963,446.314,174.076,18.270,153.042
C05079=1084.071,-72.714,446.303,174.077,18.272,153.042
C05080=1084.078,-72.464,446.292,174.079,18.273,153.042
C05081=1084.084,-72.214,446.281,174.080,18.274,153.042
C05082=1084.089,-71.965,446.270,174.082,18.276,153.042
C05083=1084.096,-71.714,446.259,174.083,18.278,153.042
C05084=1084.101,-71.465,446.248,174.084,18.279,153.042
C05085=1084.107,-71.215,446.237,174.086,18.280,153.042
C05086=1084.113,-70.966,446.226,174.087,18.282,153.042
C05087=1084.119,-70.716,446.215,174.089,18.283,153.042
C05088=1084.125,-70.466,446.204,174.090,18.285,153.042
C05089=1084.131,-70.217,446.193,174.092,18.286,153.042
C05090=1084.137,-69.967,446.182,174.093,18.287,153.042
C05091=1084.142,-69.717,446.170,174.095,18.289,153.042
C05092=1084.148,-69.468,446.159,174.096,18.291,153.042
C05093=1084.154,-69.218,446.147,174.098,18.292,153.042
C05094=1084.160,-68.968,446.137,174.099,18.293,153.042
C05095=1084.166,-68.719,446.126,174.101,18.295,153.042
C05096=1084.172,-68.468,446.114,174.102,18.296,153.042
C05097=1084.178,-68.219,446.104,174.104,18.298,153.042
C05098=1084.184,-67.970,446.092,174.105,18.299,153.042
C05099=1084.190,-67.720,446.081,174.107,18.300,153.042
C05100=1084.195,-67.470,446.069,174.108,18.302,153.042
C05101=1084.201,-67.221,446.058,174.109,18.303,153.042
C05102=1084.207,-66.970,446.047,174.111,18.305,153.042
C05103=1084.213,-66.721,446.036,174.113,18.306,153.042
C05104=1084.220,-66.471,446.024,174.114,18.308,153.042
C05105=1084.226,-66.222,446.013,174.116,18.310,153.042
C05106=1084.231,-65.972,446.003,174.118,18.311,153.042
C05107=1084.237,-65.722,445.991,174.119,18.313,153.042
C05108=1084.243,-65.448,445.978,174.121,18.314,153.042
C05109=1084.250,-65.175,445.966,174.122,18.316,153.042
C05110=1084.257,-64.901,445.954,174.124,18.317,153.042
C05111=1084.264,-64.628,445.941,174.125,18.318,153.042
C05112=1084.269,-64.378,445.930,174.127,18.321,153.042
C05113=1084.275,-64.128,445.919,174.129,18.322,153.042
C05114=1084.281,-63.878,445.908,174.130,18.324,153.042
C05115=1084.287,-63.629,445.896,174.132,18.325,153.042
C05116=1084.293,-63.379,445.885,174.133,18.327,153.042
C05117=1084.300,-63.129,445.874,174.135,18.328,153.042
C05118=1084.305,-62.880,445.861,174.136,18.329,153.042
C05119=1084.311,-62.630,445.851,174.137,18.331,153.042
C05120=1084.317,-62.380,445.839,174.139,18.332,153.042
C05121=1084.323,-62.131,445.828,174.140,18.334,153.042
C05122=1084.329,-61.881,445.816,174.142,18.336,153.042
C05123=1084.334,-61.631,445.805,174.143,18.337,153.042
C05124=1084.341,-61.382,445.793,174.145,18.338,153.042
C05125=1084.347,-61.132,445.782,174.146,18.340,153.042
C05126=1084.353,-60.882,445.771,174.148,18.341,153.042
C05127=1084.359,-60.633,445.759,174.149,18.343,153.042
C05128=1084.365,-60.383,445.748,174.150,18.344,153.042
C05129=1084.370,-60.133,445.737,174.152,18.346,153.042
C05130=1084.377,-59.884,445.725,174.154,18.347,153.042
C05131=1084.383,-59.634,445.714,174.155,18.348,153.042
C05132=1084.389,-59.384,445.703,174.156,18.350,153.042
C05133=1084.394,-59.135,445.690,174.158,18.352,153.042
C05134=1084.401,-58.884,445.679,174.159,18.353,153.042
C05135=1084.407,-58.636,445.668,174.161,18.355,153.042
C05136=1084.413,-58.385,445.656,174.163,18.357,153.043
C05137=1084.419,-58.136,445.644,174.164,18.358,153.043
C05138=1084.425,-57.886,445.633,174.166,18.360,153.043
C05139=1084.431,-57.637,445.622,174.167,18.361,153.042
C05140=1084.437,-57.387,445.610,174.169,18.362,153.043
C05141=1084.442,-57.137,445.599,174.170,18.364,153.043
C05142=1084.449,-56.888,445.587,174.172,18.365,153.043
C05143=1084.455,-56.638,445.576,174.173,18.367,153.043
C05144=1084.461,-56.389,445.564,174.175,18.369,153.043
C05145=1084.466,-56.139,445.552,174.176,18.370,153.043
C05146=1084.473,-55.889,445.540,174.177,18.372,153.043
C05147=1084.479,-55.639,445.529,174.179,18.373,153.043
C05148=1084.485,-55.390,445.517,174.180,18.374,153.043
C05149=1084.491,-55.140,445.506,174.182,18.376,153.043
C05150=1084.497,-54.891,445.494,174.183,18.377,153.043
C05151=1084.503,-54.641,445.483,174.186,18.379,153.043
C05152=1084.509,-54.391,445.471,174.187,18.381,153.043
C05153=1084.515,-54.141,445.459,174.188,18.383,153.043
C05154=1084.522,-53.892,445.447,174.190,18.384,153.043
C05155=1084.528,-53.643,445.436,174.191,18.386,153.043
C05156=1084.533,-53.392,445.424,174.193,18.387,153.043
C05157=1084.539,-53.143,445.412,174.194,18.389,153.043
C05158=1084.546,-52.893,445.401,174.195,18.390,153.043
C05159=1084.552,-52.643,445.389,174.197,18.392,153.043
C05160=1084.557,-52.394,445.378,174.199,18.393,153.043
C05161=1084.564,-52.144,445.366,174.200,18.394,153.043
C05162=1084.570,-51.895,445.354,174.201,18.396,153.043
C05163=1084.576,-51.645,445.342,174.203,18.398,153.043
C05164=1084.582,-51.395,445.330,174.205,18.400,153.043
C05165=1084.588,-51.146,445.319,174.207,18.401,153.043
C05166=1084.594,-50.896,445.307,174.208,18.403,153.043
C05167=1084.601,-50.646,445.295,174.209,18.404,153.043
C05168=1084.606,-50.397,445.284,174.211,18.406,153.043
C05169=1084.612,-50.147,445.272,174.212,18.407,153.043
C05170=1084.617,-49.898,445.259,174.214,18.409,153.043
C05171=1084.624,-49.648,445.248,174.215,18.410,153.043
C05172=1084.631,-49.375,445.234,174.216,18.412,153.043
C05173=1084.637,-49.103,445.222,174.218,18.415,153.043
C05174=1084.643,-48.830,445.209,174.220,18.416,153.043
C05175=1084.650,-48.558,445.196,174.221,18.418,153.043
C05176=1084.655,-48.308,445.184,174.223,18.419,153.044
C05177=1084.661,-48.059,445.172,174.224,18.421,153.044
C05178=1084.667,-47.809,445.160,174.226,18.423,153.044
C05179=1084.673,-47.560,445.149,174.228,18.424,153.044
C05180=1084.679,-47.310,445.136,174.229,18.426,153.044
C05181=1084.685,-47.060,445.124,174.231,18.427,153.044
C05182=1084.691,-46.811,445.112,174.232,18.429,153.044
C05183=1084.696,-46.560,445.100,174.233,18.431,153.044
C05184=1084.703,-46.311,445.088,174.235,18.433,153.044
C05185=1084.708,-46.062,445.076,174.236,18.434,153.044
C05186=1084.714,-45.812,445.064,174.237,18.436,153.044
C05187=1084.720,-45.562,445.053,174.240,18.438,153.044
C05188=1084.726,-45.312,445.040,174.241,18.439,153.044
C05189=1084.733,-45.063,445.028,174.243,18.441,153.044
C05190=1084.738,-44.814,445.016,174.244,18.442,153.044
C05191=1084.744,-44.564,445.003,174.245,18.444,153.044
C05192=1084.750,-44.314,444.992,174.247,18.446,153.044
C05193=1084.755,-44.064,444.980,174.248,18.447,153.044
C05194=1084.762,-43.815,444.968,174.249,18.449,153.044
C05195=1084.768,-43.565,444.955,174.251,18.451,153.044
C05196=1084.773,-43.316,444.943,174.253,18.453,153.044
C05197=1084.780,-43.066,444.932,174.255,18.454,153.044
C05198=1084.786,-42.816,444.920,174.256,18.456,153.044
C05199=1084.791,-42.567,444.907,174.257,18.457,153.045
C05200=1084.798,-42.317,444.895,174.259,18.459,153.045
C05201=1084.803,-42.067,444.883,174.260,18.460,153.045
C05202=1084.809,-41.818,444.871,174.262,18.462,153.045
C05203=1084.815,-41.568,444.859,174.263,18.464,153.045
C05204=1084.821,-41.318,444.846,174.265,18.466,153.045
C05205=1084.826,-41.069,444.835,174.267,18.468,153.045
C05206=1084.833,-40.819,444.823,174.268,18.469,153.045
C05207=1084.839,-40.569,444.810,174.269,18.471,153.045
C05208=1084.845,-40.320,444.798,174.271,18.472,153.045
C05209=1084.851,-40.070,444.786,174.272,18.474,153.045
C05210=1084.857,-39.821,444.773,174.274,18.475,153.045
C05211=1084.863,-39.571,444.761,174.275,18.477,153.045
C05212=1084.869,-39.321,444.749,174.277,18.480,153.045
C05213=1084.875,-39.072,444.737,174.278,18.481,153.045
C05214=1084.880,-38.822,444.724,174.280,18.483,153.045
C05215=1084.887,-38.572,444.712,174.281,18.484,153.045
C05216=1084.892,-38.323,444.700,174.283,18.486,153.045
C05217=1084.898,-38.073,444.687,174.284,18.487,153.045
C05218=1084.904,-37.824,444.675,174.285,18.489,153.046
C05219=1084.910,-37.574,444.662,174.288,18.491,153.046
C05220=1084.916,-37.325,444.651,174.289,18.493,153.046
C05221=1084.922,-37.075,444.638,174.290,18.495,153.046
C05222=1084.928,-36.825,444.626,174.292,18.496,153.046
C05223=1084.933,-36.576,444.613,174.293,18.498,153.046
C05224=1084.939,-36.326,444.601,174.294,18.500,153.046
C05225=1084.945,-36.076,444.588,174.296,18.501,153.046
C05226=1084.951,-35.826,444.576,174.298,18.503,153.046
C05227=1084.957,-35.577,444.564,174.300,18.505,153.046
C05228=1084.963,-35.327,444.552,174.301,18.507,153.046
C05229=1084.969,-35.078,444.539,174.302,18.508,153.046
C05230=1084.975,-34.828,444.527,174.304,18.510,153.046
C05231=1084.980,-34.578,444.514,174.305,18.512,153.046
C05232=1084.986,-34.329,444.502,174.306,18.514,153.046
C05233=1084.992,-34.079,444.489,174.308,18.516,153.046
C05234=1084.998,-33.829,444.476,174.310,18.517,153.047
C05235=1085.004,-33.581,444.464,174.311,18.519,153.047
C05236=1085.010,-33.308,444.450,174.312,18.521,153.047
C05237=1085.017,-33.036,444.437,174.315,18.523,153.047
C05238=1085.024,-32.764,444.423,174.316,18.524,153.047
C05239=1085.029,-32.492,444.409,174.317,18.526,153.047
C05240=1085.036,-32.242,444.397,174.319,18.528,153.047
C05241=1085.042,-31.992,444.385,174.321,18.530,153.047
C05242=1085.048,-31.743,444.372,174.322,18.532,153.047
C05243=1085.054,-31.493,444.360,174.324,18.533,153.047
C05244=1085.059,-31.244,444.348,174.325,18.535,153.047
C05245=1085.065,-30.994,444.334,174.326,18.537,153.047
C05246=1085.071,-30.744,444.322,174.328,18.538,153.047
C05247=1085.077,-30.495,444.309,174.330,18.540,153.047
C05248=1085.083,-30.245,444.297,174.331,18.542,153.047
C05249=1085.089,-29.995,444.284,174.333,18.544,153.048
C05250=1085.094,-29.746,444.271,174.334,18.546,153.048
C05251=1085.100,-29.496,444.259,174.336,18.547,153.048
C05252=1085.106,-29.246,444.246,174.337,18.549,153.048
C05253=1085.112,-28.997,444.233,174.339,18.551,153.048
C05254=1085.119,-28.748,444.221,174.340,18.553,153.048
C05255=1085.125,-28.498,444.208,174.342,18.554,153.048
C05256=1085.130,-28.249,444.196,174.343,18.556,153.048
C05257=1085.136,-27.999,444.183,174.344,18.558,153.048
C05258=1085.142,-27.749,444.170,174.346,18.559,153.048
C05259=1085.148,-27.499,444.158,174.348,18.561,153.048
C05260=1085.154,-27.250,444.145,174.350,18.563,153.048
C05261=1085.160,-27.000,444.132,174.351,18.565,153.048
C05262=1085.166,-26.750,444.119,174.352,18.567,153.048
C05263=1085.172,-26.501,444.107,174.354,18.568,153.048
C05264=1085.178,-26.251,444.095,174.356,18.571,153.049
C05265=1085.183,-26.002,444.081,174.357,18.572,153.049
C05266=1085.189,-25.752,444.068,174.358,18.574,153.049
C05267=1085.195,-25.502,444.056,174.360,18.576,153.049
C05268=1085.201,-25.253,444.042,174.361,18.577,153.049
C05269=1085.207,-25.003,444.030,174.362,18.579,153.049
C05270=1085.213,-24.754,444.017,174.365,18.581,153.049
C05271=1085.218,-24.504,444.004,174.366,18.583,153.049
C05272=1085.224,-24.254,443.991,174.367,18.585,153.049
C05273=1085.230,-24.005,443.978,174.369,18.586,153.049
C05274=1085.236,-23.755,443.965,174.370,18.588,153.049
C05275=1085.242,-23.505,443.953,174.372,18.590,153.049
C05276=1085.248,-23.256,443.940,174.374,18.592,153.049
C05277=1085.254,-23.006,443.927,174.375,18.594,153.050
C05278=1085.259,-22.757,443.913,174.376,18.595,153.050
C05279=1085.265,-22.507,443.901,174.378,18.597,153.050
C05280=1085.271,-22.258,443.888,174.380,18.600,153.050
C05281=1085.277,-22.008,443.875,174.381,18.601,153.050
C05282=1085.283,-21.758,443.863,174.382,18.603,153.050
C05283=1085.289,-21.509,443.849,174.384,18.605,153.050
C05284=1085.294,-21.259,443.836,174.385,18.606,153.050
C05285=1085.300,-21.010,443.823,174.387,18.608,153.050
C05286=1085.306,-20.760,443.810,174.389,18.610,153.050
C05287=1085.312,-20.510,443.797,174.390,18.612,153.050
C05288=1085.318,-20.261,443.784,174.391,18.613,153.050
C05289=1085.324,-20.011,443.771,174.393,18.616,153.051
C05290=1085.329,-19.762,443.758,174.395,18.618,153.051
C05291=1085.335,-19.513,443.745,174.396,18.619,153.051
C05292=1085.341,-19.263,443.733,174.397,18.621,153.051
C05293=1085.347,-19.013,443.719,174.399,18.623,153.051
C05294=1085.353,-18.763,443.706,174.400,18.624,153.051
C05295=1085.359,-18.514,443.693,174.402,18.627,153.051
C05296=1085.365,-18.264,443.680,174.404,18.628,153.051
C05297=1085.371,-18.015,443.667,174.405,18.630,153.051
C05298=1085.376,-17.765,443.653,174.407,18.631,153.051
C05299=1085.382,-17.515,443.641,174.408,18.633,153.051
C05300=1085.389,-17.242,443.626,174.410,18.636,153.051
C05301=1085.395,-16.969,443.612,174.411,18.638,153.051
C05302=1085.401,-16.697,443.598,174.413,18.640,153.051
C05303=1085.408,-16.423,443.583,174.415,18.642,153.052
C05304=1085.414,-16.174,443.570,174.416,18.643,153.052
C05305=1085.420,-15.924,443.557,174.417,18.645,153.052
C05306=1085.426,-15.675,443.544,174.419,18.647,153.052
C05307=1085.432,-15.425,443.530,174.421,18.649,153.052
C05308=1085.438,-15.175,443.517,174.422,18.650,153.052
C05309=1085.444,-14.926,443.504,174.424,18.653,153.052
C05310=1085.450,-14.677,443.490,174.426,18.655,153.052
C05311=1085.455,-14.427,443.478,174.427,18.656,153.052
C05312=1085.462,-14.177,443.464,174.428,18.658,153.052
C05313=1085.467,-13.928,443.451,174.430,18.660,153.052
C05314=1085.473,-13.678,443.438,174.431,18.661,153.052
C05315=1085.479,-13.428,443.424,174.433,18.664,153.053
C05316=1085.485,-13.179,443.411,174.435,18.665,153.053
C05317=1085.490,-12.929,443.398,174.436,18.667,153.053
C05318=1085.496,-12.680,443.384,174.437,18.669,153.053
C05319=1085.502,-12.430,443.371,174.440,18.671,153.053
C05320=1085.508,-12.180,443.358,174.441,18.673,153.053
C05321=1085.514,-11.931,443.345,174.442,18.675,153.053
C05322=1085.519,-11.681,443.331,174.443,18.677,153.053
C05323=1085.525,-11.432,443.318,174.445,18.678,153.053
C05324=1085.531,-11.182,443.305,174.447,18.680,153.053
C05325=1085.537,-10.933,443.291,174.448,18.682,153.053
C05326=1085.542,-10.683,443.277,174.450,18.684,153.053
C05327=1085.549,-10.434,443.264,174.451,18.686,153.054
C05328=1085.555,-10.184,443.251,174.453,18.688,153.054
C05329=1085.560,-9.934,443.238,174.455,18.689,153.054
C05330=1085.566,-9.685,443.224,174.456,18.692,153.054
C05331=1085.572,-9.435,443.211,174.457,18.693,153.054
C05332=1085.578,-9.186,443.197,174.459,18.696,153.054
C05333=1085.583,-8.937,443.183,174.461,18.697,153.054
C05334=1085.589,-8.687,443.171,174.462,18.699,153.054
C05335=1085.595,-8.437,443.157,174.463,18.701,153.054
C05336=1085.601,-8.188,443.144,174.465,18.703,153.054
C05337=1085.607,-7.938,443.130,174.467,18.704,153.054
C05338=1085.613,-7.688,443.116,174.468,18.706,153.055
C05339=1085.619,-7.439,443.102,174.469,18.708,153.055
C05340=1085.625,-7.190,443.089,174.471,18.710,153.055
C05341=1085.630,-6.939,443.076,174.473,18.712,153.055
C05342=1085.636,-6.690,443.063,174.474,18.714,153.055
C05343=1085.642,-6.440,443.049,174.476,18.716,153.055
C05344=1085.648,-6.191,443.036,174.477,18.717,153.055
C05345=1085.653,-5.942,443.022,174.479,18.719,153.055
C05346=1085.660,-5.692,443.008,174.480,18.721,153.055
C05347=1085.666,-5.442,442.994,174.482,18.723,153.055
C05348=1085.672,-5.193,442.981,174.483,18.725,153.055
C05349=1085.677,-4.943,442.967,174.485,18.727,153.055
C05350=1085.683,-4.694,442.953,174.487,18.728,153.055
C05351=1085.689,-4.444,442.940,174.488,18.731,153.056
C05352=1085.695,-4.195,442.926,174.489,18.732,153.056
C05353=1085.701,-3.945,442.912,174.492,18.734,153.056
C05354=1085.707,-3.695,442.899,174.493,18.736,153.056
C05355=1085.713,-3.446,442.885,174.494,18.738,153.056
C05356=1085.719,-3.196,442.871,174.495,18.740,153.056
C05357=1085.724,-2.947,442.858,174.498,18.742,153.056
C05358=1085.730,-2.698,442.844,174.499,18.743,153.056
C05359=1085.736,-2.448,442.830,174.500,18.745,153.056
C05360=1085.741,-2.198,442.817,174.502,18.747,153.056
C05361=1085.747,-1.949,442.803,174.504,18.750,153.057
C05362=1085.753,-1.699,442.789,174.505,18.751,153.057
C05363=1085.759,-1.449,442.775,174.506,18.753,153.057
C05364=1085.765,-1.175,442.761,174.509,18.755,153.057
C05365=1085.771,-0.901,442.745,174.510,18.757,153.057
C05366=1085.778,-0.626,442.730,174.512,18.760,153.057
C05367=1085.784,-0.351,442.715,174.513,18.761,153.057
C05368=1085.790,-0.102,442.701,174.514,18.763,153.057
C05369=1085.795,0.148,442.687,174.517,18.765,153.057
C05370=1085.801,0.398,442.673,174.518,18.767,153.057
C05371=1085.806,0.647,442.659,174.519,18.769,153.058
C05372=1085.813,0.897,442.646,174.521,18.772,153.058
C05373=1085.818,1.147,442.632,174.523,18.773,153.058
C05374=1085.824,1.396,442.617,174.524,18.775,153.058
C05375=1085.830,1.645,442.603,174.525,18.777,153.058
C05376=1085.835,1.895,442.589,174.528,18.779,153.058
C05377=1085.841,2.144,442.576,174.529,18.781,153.058
C05378=1085.847,2.394,442.562,174.530,18.782,153.058
C05379=1085.853,2.644,442.548,174.531,18.784,153.058
C05380=1085.858,2.893,442.534,174.534,18.786,153.058
C05381=1085.864,3.142,442.520,174.535,18.788,153.059
C05382=1085.870,3.392,442.506,174.536,18.790,153.059
C05383=1085.877,3.642,442.492,174.539,18.792,153.059
C05384=1085.882,3.892,442.478,174.540,18.794,153.059
C05385=1085.887,4.141,442.464,174.541,18.796,153.059
C05386=1085.893,4.390,442.450,174.542,18.798,153.059
C05387=1085.899,4.640,442.436,174.545,18.800,153.059
C05388=1085.905,4.890,442.422,174.546,18.802,153.059
C05389=1085.911,5.139,442.408,174.547,18.803,153.059
C05390=1085.917,5.388,442.394,174.549,18.805,153.059
C05391=1085.922,5.638,442.380,174.551,18.807,153.059
C05392=1085.928,5.888,442.366,174.552,18.809,153.059
C05393=1085.934,6.138,442.352,174.553,18.811,153.060
C05394=1085.940,6.387,442.337,174.556,18.813,153.060
C05395=1085.945,6.636,442.323,174.557,18.815,153.060
C05396=1085.951,6.886,442.309,174.558,18.817,153.060
C05397=1085.958,7.135,442.295,174.560,18.818,153.060
C05398=1085.963,7.385,442.281,174.562,18.821,153.060
C05399=1085.969,7.634,442.268,174.563,18.822,153.060
C05400=1085.975,7.884,442.253,174.564,18.824,153.060
C05401=1085.981,8.133,442.239,174.567,18.826,153.060
C05402=1085.986,8.383,442.225,174.568,18.828,153.060
C05403=1085.992,8.633,442.210,174.569,18.830,153.060
C05404=1085.998,8.882,442.196,174.571,18.831,153.061
C05405=1086.003,9.132,442.182,174.573,18.834,153.061
C05406=1086.010,9.381,442.168,174.574,18.836,153.061
C05407=1086.016,9.631,442.154,174.576,18.837,153.061
C05408=1086.021,9.880,442.140,174.578,18.840,153.061
C05409=1086.027,10.129,442.126,174.579,18.841,153.061
C05410=1086.033,10.380,442.111,174.580,18.843,153.061
C05411=1086.039,10.628,442.097,174.582,18.845,153.061
C05412=1086.045,10.878,442.083,174.584,18.847,153.061
C05413=1086.051,11.128,442.069,174.585,18.849,153.061
C05414=1086.056,11.377,442.054,174.587,18.850,153.061
C05415=1086.062,11.628,442.040,174.589,18.852,153.061
C05416=1086.068,11.876,442.025,174.590,18.854,153.062
C05417=1086.074,12.126,442.011,174.591,18.856,153.062
C05418=1086.080,12.376,441.996,174.593,18.859,153.062
C05419=1086.086,12.625,441.983,174.595,18.860,153.062
C05420=1086.092,12.874,441.969,174.596,18.862,153.062
C05421=1086.098,13.124,441.954,174.598,18.864,153.062
C05422=1086.104,13.373,441.940,174.600,18.866,153.062
C05423=1086.110,13.623,441.926,174.601,18.867,153.062
C05424=1086.116,13.872,441.911,174.602,18.869,153.062
C05425=1086.121,14.122,441.897,174.605,18.871,153.062
C05426=1086.128,14.372,441.882,174.606,18.873,153.062
C05427=1086.133,14.621,441.868,174.607,18.875,153.062
C05428=1086.140,14.898,441.852,174.609,18.877,153.063
C05429=1086.145,15.174,441.836,174.611,18.879,153.063
C05430=1086.152,15.451,441.819,174.613,18.882,153.063
C05431=1086.158,15.727,441.804,174.614,18.883,153.063
C05432=1086.164,15.978,441.789,174.616,18.886,153.063
C05433=1086.170,16.226,441.775,174.618,18.887,153.063
C05434=1086.176,16.475,441.760,174.619,18.889,153.063
C05435=1086.182,16.726,441.746,174.621,18.891,153.063
C05436=1086.187,16.975,441.731,174.623,18.893,153.063
C05437=1086.193,17.225,441.717,174.624,18.895,153.063
C05438=1086.199,17.474,441.702,174.626,18.897,153.063
C05439=1086.205,17.723,441.687,174.627,18.899,153.064
C05440=1086.211,17.973,441.673,174.629,18.900,153.064
C05441=1086.217,18.222,441.659,174.631,18.903,153.064
C05442=1086.222,18.472,441.643,174.632,18.905,153.064
C05443=1086.228,18.722,441.629,174.634,18.906,153.064
C05444=1086.234,18.971,441.615,174.636,18.909,153.064
C05445=1086.240,19.221,441.600,174.637,18.910,153.064
C05446=1086.245,19.470,441.586,174.638,18.912,153.064
C05447=1086.252,19.720,441.571,174.641,18.914,153.064
C05448=1086.257,19.969,441.556,174.642,18.916,153.064
C05449=1086.262,20.219,441.542,174.643,18.918,153.065
C05450=1086.269,20.468,441.527,174.645,18.920,153.065
C05451=1086.274,20.717,441.512,174.647,18.921,153.065
C05452=1086.280,20.967,441.497,174.648,18.923,153.065
C05453=1086.286,21.217,441.483,174.650,18.926,153.065
C05454=1086.291,21.466,441.468,174.652,18.928,153.065
C05455=1086.298,21.715,441.453,174.653,18.929,153.065
C05456=1086.303,21.965,441.438,174.654,18.931,153.065
